LIN {X 0.124,Y -428.626,Z 670.577,A 0.000,B 0.000,C 90.000,E1 103.883} C_DIS
LIN {X -0.109,Y -448.565,Z 670.566,A 0.000,B 0.000,C 90.000,E1 101.827} C_DIS
LIN {X -0.065,Y -469.090,Z 670.555,A 0.000,B 0.000,C 90.000,E1 99.905} C_DIS
LIN {X -0.014,Y -471.282,Z 670.554,A 0.000,B 0.000,C 90.000,E1 99.670} C_DIS
LIN {X -0.163,Y -473.093,Z 670.552,A 0.000,B 0.000,C 90.000,E1 99.434} C_DIS
LIN {X 0.078,Y -474.453,Z 670.551,A 0.000,B 0.000,C 90.000,E1 99.151} C_DIS
LIN {X -0.202,Y -476.161,Z 670.548,A 0.000,B 0.000,C 90.000,E1 98.681} C_DIS
LIN {X -0.076,Y -476.795,Z 670.545,A 0.000,B 0.000,C 90.000,E1 98.163} C_DIS
LIN {X 0.062,Y -476.462,Z 670.542,A 0.000,B 0.000,C 90.000,E1 97.644} C_DIS
LIN {X 0.204,Y -475.113,Z 670.540,A 0.000,B 0.000,C 90.000,E1 97.125} C_DIS
LIN {X 0.067,Y -473.992,Z 670.538,A 0.000,B 0.000,C 90.000,E1 96.891} C_DIS
LIN {X -0.126,Y -472.493,Z 670.537,A 0.000,B 0.000,C 90.000,E1 96.663} C_DIS
LIN {X -0.192,Y -455.641,Z 670.523,A 0.000,B 0.000,C 90.000,E1 94.131} C_DIS
LIN {X 0.189,Y -443.555,Z 670.511,A 0.000,B 0.000,C 90.000,E1 92.007} C_DIS
LIN {X 0.104,Y -433.501,Z 670.501,A 0.000,B 0.000,C 90.000,E1 90.172} C_DIS
LIN {X -0.022,Y -425.963,Z 670.494,A 0.000,B 0.000,C 90.000,E1 88.854} C_DIS
LIN {X -0.041,Y -415.056,Z 670.483,A 0.000,B 0.000,C 90.000,E1 86.963} C_DIS
LIN {X 0.179,Y -404.176,Z 670.472,A 0.000,B 0.000,C 90.000,E1 85.008} C_DIS
LIN {X -0.101,Y -390.407,Z 670.458,A 0.000,B 0.000,C 90.000,E1 82.527} C_DIS
LIN {X 0.116,Y -378.549,Z 670.446,A 0.000,B 0.000,C 90.000,E1 80.208} C_DIS
LIN {X 0.087,Y -365.737,Z 670.431,A 0.000,B 0.000,C 90.000,E1 77.589} C_DIS
LIN {X -0.091,Y -350.683,Z 670.413,A 0.000,B 0.000,C 90.000,E1 74.338} C_DIS
LIN {X -0.019,Y -337.744,Z 670.396,A 0.000,B 0.000,C 90.000,E1 71.275} C_DIS
LIN {X -0.086,Y -323.394,Z 670.375,A 0.000,B 0.000,C 90.000,E1 67.539} C_DIS
LIN {X -0.074,Y -311.579,Z 670.356,A 0.000,B 0.000,C 90.000,E1 64.024} C_DIS
LIN {X -0.193,Y -301.989,Z 670.338,A 0.000,B 0.000,C 90.000,E1 60.795} C_DIS
LIN {X -0.016,Y -293.247,Z 670.319,A 0.000,B 0.000,C 90.000,E1 57.454} C_DIS
LIN {X -0.007,Y -286.662,Z 670.304,A 0.000,B 0.000,C 90.000,E1 54.769} C_DIS
LIN {X -0.067,Y -280.101,Z 670.289,A 0.000,B 0.000,C 90.000,E1 52.065} C_DIS
LIN {X 0.013,Y -274.939,Z 670.278,A 0.000,B 0.000,C 90.000,E1 49.989} C_DIS
LIN {X -0.032,Y -269.443,Z 670.266,A 0.000,B 0.000,C 90.000,E1 47.919} C_DIS
LIN {X 0.004,Y -263.583,Z 670.255,A 0.000,B 0.000,C 90.000,E1 45.810} C_DIS
LIN {X -0.079,Y -257.402,Z 670.243,A 0.000,B 0.000,C 90.000,E1 43.704} C_DIS
LIN {X 0.092,Y -251.028,Z 670.231,A 0.000,B 0.000,C 90.000,E1 41.515} C_DIS
LIN {X 0.007,Y -242.450,Z 670.215,A 0.000,B 0.000,C 90.000,E1 38.624} C_DIS
LIN {X 0.081,Y -232.462,Z 670.194,A 0.000,B 0.000,C 90.000,E1 34.898} C_DIS
LIN {X 0.078,Y -225.134,Z 670.177,A 0.000,B 0.000,C 90.000,E1 31.878} C_DIS
LIN {X 0.042,Y -218.649,Z 670.160,A 0.000,B 0.000,C 90.000,E1 28.821} C_DIS
LIN {X 0.018,Y -212.967,Z 670.143,A 0.000,B 0.000,C 90.000,E1 25.720} C_DIS
LIN {X -0.032,Y -208.075,Z 670.125,A 0.000,B 0.000,C 90.000,E1 22.589} C_DIS
LIN {X 0.022,Y -203.111,Z 670.103,A 0.000,B 0.000,C 90.000,E1 18.598} C_DIS
LIN {X -0.017,Y -199.233,Z 670.081,A 0.000,B 0.000,C 90.000,E1 14.592} C_DIS
LIN {X -0.006,Y -195.919,Z 670.054,A 0.000,B 0.000,C 90.000,E1 9.726} C_DIS
LIN {X 0.082,Y -193.629,Z 670.013,A 0.000,B 0.000,C 90.000,E1 2.350} C_DIS
LIN {X -0.036,Y -195.477,Z 669.961,A 0.000,B 0.000,C 90.000,E1 352.996} C_DIS
LIN {X -0.065,Y -198.507,Z 669.934,A 0.000,B 0.000,C 90.000,E1 348.117} C_DIS
LIN {X 0.026,Y -202.213,Z 669.911,A 0.000,B 0.000,C 90.000,E1 344.047} C_DIS
LIN {X -0.061,Y -206.877,Z 669.889,A 0.000,B 0.000,C 90.000,E1 340.061} C_DIS
LIN {X 0.099,Y -212.320,Z 669.867,A 0.000,B 0.000,C 90.000,E1 336.049} C_DIS
LIN {X 0.007,Y -218.539,Z 669.845,A 0.000,B 0.000,C 90.000,E1 332.153} C_DIS
LIN {X 0.029,Y -225.425,Z 669.824,A 0.000,B 0.000,C 90.000,E1 328.280} C_DIS
LIN {X -0.027,Y -232.928,Z 669.803,A 0.000,B 0.000,C 90.000,E1 324.482} C_DIS
LIN {X 0.003,Y -241.051,Z 669.782,A 0.000,B 0.000,C 90.000,E1 320.723} C_DIS
LIN {X 0.037,Y -250.012,Z 669.761,A 0.000,B 0.000,C 90.000,E1 317.025} C_DIS
LIN {X -0.054,Y -259.057,Z 669.743,A 0.000,B 0.000,C 90.000,E1 313.785} C_DIS
LIN {X 0.029,Y -270.150,Z 669.723,A 0.000,B 0.000,C 90.000,E1 310.216} C_DIS
LIN {X 0.081,Y -281.443,Z 669.706,A 0.000,B 0.000,C 90.000,E1 307.076} C_DIS
LIN {X -0.056,Y -295.332,Z 669.687,A 0.000,B 0.000,C 90.000,E1 303.706} C_DIS
LIN {X 0.006,Y -310.666,Z 669.669,A 0.000,B 0.000,C 90.000,E1 300.384} C_DIS
LIN {X -0.071,Y -327.476,Z 669.651,A 0.000,B 0.000,C 90.000,E1 297.180} C_DIS
LIN {X 0.104,Y -341.711,Z 669.637,A 0.000,B 0.000,C 90.000,E1 294.643} C_DIS
LIN {X 0.144,Y -360.271,Z 669.620,A 0.000,B 0.000,C 90.000,E1 291.589} C_DIS
LIN {X 0.097,Y -372.192,Z 669.610,A 0.000,B 0.000,C 90.000,E1 289.812} C_DIS
LIN {X -0.071,Y -389.779,Z 669.597,A 0.000,B 0.000,C 90.000,E1 287.511} C_DIS
LIN {X -0.123,Y -406.148,Z 669.586,A 0.000,B 0.000,C 90.000,E1 285.536} C_DIS
LIN {X 0.094,Y -417.666,Z 669.578,A 0.000,B 0.000,C 90.000,E1 284.120} C_DIS
LIN {X -0.167,Y -426.483,Z 669.572,A 0.000,B 0.000,C 90.000,E1 283.063} C_DIS
LIN {X -0.137,Y -437.045,Z 669.565,A 0.000,B 0.000,C 90.000,E1 281.715} C_DIS
LIN {X -0.177,Y -445.024,Z 669.559,A 0.000,B 0.000,C 90.000,E1 280.658} C_DIS
LIN {X -0.112,Y -465.214,Z 669.545,A 0.000,B 0.000,C 90.000,E1 278.049} C_DIS
LIN {X -0.217,Y -470.973,Z 669.540,A 0.000,B 0.000,C 90.000,E1 277.296} C_DIS
LIN {X -0.120,Y -474.369,Z 669.538,A 0.000,B 0.000,C 90.000,E1 276.777} C_DIS
LIN {X -0.144,Y -478.628,Z 669.533,A 0.000,B 0.000,C 90.000,E1 276.024} C_DIS
LIN {X -0.047,Y -481.033,Z 669.531,A 0.000,B 0.000,C 90.000,E1 275.511} C_DIS
LIN {X -0.020,Y -483.884,Z 669.526,A 0.000,B 0.000,C 90.000,E1 274.759} C_DIS
LIN {X 0.114,Y -485.270,Z 669.524,A 0.000,B 0.000,C 90.000,E1 274.245} C_DIS
LIN {X -0.187,Y -486.308,Z 669.521,A 0.000,B 0.000,C 90.000,E1 273.784} C_DIS
LIN {X -0.028,Y -486.967,Z 669.518,A 0.000,B 0.000,C 90.000,E1 273.269} C_DIS
LIN {X 0.167,Y -487.304,Z 669.515,A 0.000,B 0.000,C 90.000,E1 272.751} C_DIS
LIN {X -0.146,Y -487.303,Z 669.513,A 0.000,B 0.000,C 90.000,E1 272.293} C_DIS
LIN {X 0.048,Y -487.013,Z 669.510,A 0.000,B 0.000,C 90.000,E1 271.776} C_DIS
LIN {X 0.224,Y -486.400,Z 669.507,A 0.000,B 0.000,C 90.000,E1 271.260} C_DIS
LIN {X -0.086,Y -485.361,Z 669.504,A 0.000,B 0.000,C 90.000,E1 270.802} C_DIS
LIN {X 0.087,Y -483.834,Z 669.502,A 0.000,B 0.000,C 90.000,E1 270.286} C_DIS
LIN {X -0.228,Y -481.687,Z 669.499,A 0.000,B 0.000,C 90.000,E1 269.828} C_DIS
LIN {X -0.070,Y -478.880,Z 669.496,A 0.000,B 0.000,C 90.000,E1 269.312} C_DIS
LIN {X 0.066,Y -475.210,Z 669.493,A 0.000,B 0.000,C 90.000,E1 268.797} C_DIS
LIN {X -0.113,Y -473.058,Z 669.492,A 0.000,B 0.000,C 90.000,E1 268.568} C_DIS
LIN {X 0.039,Y -467.847,Z 669.489,A 0.000,B 0.000,C 90.000,E1 268.051} C_DIS
LIN {X -0.115,Y -464.818,Z 669.488,A 0.000,B 0.000,C 90.000,E1 267.822} C_DIS
LIN {X 0.064,Y -458.384,Z 669.485,A 0.000,B 0.000,C 90.000,E1 267.364} C_DIS
LIN {X -0.102,Y -451.464,Z 669.483,A 0.000,B 0.000,C 90.000,E1 267.020} C_DIS
LIN {X -0.140,Y -444.281,Z 669.482,A 0.000,B 0.000,C 90.000,E1 266.731} C_DIS
LIN {X -0.172,Y -436.408,Z 669.480,A 0.000,B 0.000,C 90.000,E1 266.502} C_DIS
LIN {X -0.153,Y -427.882,Z 669.479,A 0.000,B 0.000,C 90.000,E1 266.331} C_DIS
LIN {X 0.061,Y -420.369,Z 669.479,A 0.000,B 0.000,C 90.000,E1 266.216} C_DIS
LIN {X -0.147,Y -413.980,Z 669.479,A 0.000,B 0.000,C 90.000,E1 266.216} C_DIS
LIN {X -0.086,Y -180.929,Z 669.479,A 0.000,B 0.000,C 90.000,E1 266.216} C_DIS
LIN {X 0.002,Y -180.904,Z 669.474,A 0.000,B 0.000,C 90.000,E1 265.298} C_DIS
LIN {X -0.048,Y -180.244,Z 669.465,A 0.000,B 0.000,C 90.000,E1 263.628} C_DIS
LIN {X -0.029,Y -178.732,Z 669.441,A 0.000,B 0.000,C 90.000,E1 259.398} C_DIS
LIN {X 0.038,Y -175.779,Z 669.413,A 0.000,B 0.000,C 90.000,E1 254.283} C_DIS
LIN {X 0.026,Y -171.963,Z 669.384,A 0.000,B 0.000,C 90.000,E1 249.156} C_DIS
LIN {X 0.063,Y -171.359,Z 669.379,A 0.000,B 0.000,C 90.000,E1 248.284} C_DIS
LIN {X 0.040,Y -167.608,Z 669.355,A 0.000,B 0.000,C 90.000,E1 243.973} C_DIS
LIN {X 0.053,Y -166.255,Z 669.346,A 0.000,B 0.000,C 90.000,E1 242.231} C_DIS
LIN {X 0.040,Y -163.009,Z 669.326,A 0.000,B 0.000,C 90.000,E1 238.742} C_DIS
LIN {X -0.046,Y -160.932,Z 669.312,A 0.000,B 0.000,C 90.000,E1 236.135} C_DIS
LIN {X 0.064,Y -157.692,Z 669.292,A 0.000,B 0.000,C 90.000,E1 232.557} C_DIS
LIN {X 0.001,Y -155.732,Z 669.277,A 0.000,B 0.000,C 90.000,E1 229.908} C_DIS
LIN {X 0.056,Y -151.990,Z 669.252,A 0.000,B 0.000,C 90.000,E1 225.405} C_DIS
LIN {X 0.071,Y -150.234,Z 669.237,A 0.000,B 0.000,C 90.000,E1 222.690} C_DIS
LIN {X -0.006,Y -146.995,Z 669.212,A 0.000,B 0.000,C 90.000,E1 218.177} C_DIS
LIN {X -0.016,Y -145.580,Z 669.197,A 0.000,B 0.000,C 90.000,E1 215.438} C_DIS
LIN {X -0.022,Y -142.969,Z 669.171,A 0.000,B 0.000,C 90.000,E1 210.846} C_DIS
LIN {X 0.032,Y -141.596,Z 669.151,A 0.000,B 0.000,C 90.000,E1 207.129} C_DIS
LIN {X -0.052,Y -139.422,Z 669.115,A 0.000,B 0.000,C 90.000,E1 200.663} C_DIS
LIN {X -0.001,Y -139.149,Z 669.104,A 0.000,B 0.000,C 90.000,E1 198.779} C_DIS
LIN {X 0.021,Y -138.346,Z 669.058,A 0.000,B 0.000,C 90.000,E1 190.366} C_DIS
LIN {X 0.006,Y -139.487,Z 669.006,A 0.000,B 0.000,C 90.000,E1 181.031} C_DIS
LIN {X -0.054,Y -141.088,Z 668.975,A 0.000,B 0.000,C 90.000,E1 175.469} C_DIS
LIN {X 0.041,Y -142.466,Z 668.959,A 0.000,B 0.000,C 90.000,E1 172.648} C_DIS
LIN {X -0.011,Y -144.711,Z 668.934,A 0.000,B 0.000,C 90.000,E1 168.049} C_DIS
LIN {X -0.060,Y -147.309,Z 668.913,A 0.000,B 0.000,C 90.000,E1 164.393} C_DIS
LIN {X -0.045,Y -150.631,Z 668.888,A 0.000,B 0.000,C 90.000,E1 159.826} C_DIS
LIN {X 0.031,Y -154.107,Z 668.868,A 0.000,B 0.000,C 90.000,E1 156.177} C_DIS
LIN {X -0.045,Y -157.530,Z 668.848,A 0.000,B 0.000,C 90.000,E1 152.615} C_DIS
LIN {X -0.100,Y -161.766,Z 668.828,A 0.000,B 0.000,C 90.000,E1 149.076} C_DIS
LIN {X 0.005,Y -165.958,Z 668.808,A 0.000,B 0.000,C 90.000,E1 145.515} C_DIS
LIN {X 0.001,Y -170.952,Z 668.789,A 0.000,B 0.000,C 90.000,E1 142.029} C_DIS
LIN {X 0.053,Y -175.820,Z 668.770,A 0.000,B 0.000,C 90.000,E1 138.566} C_DIS
LIN {X 0.048,Y -181.427,Z 668.751,A 0.000,B 0.000,C 90.000,E1 135.162} C_DIS
LIN {X -0.078,Y -186.932,Z 668.732,A 0.000,B 0.000,C 90.000,E1 131.838} C_DIS
LIN {X 0.094,Y -191.070,Z 668.720,A 0.000,B 0.000,C 90.000,E1 129.564} C_DIS
LIN {X 0.096,Y -288.280,Z 668.720,A 0.000,B 0.000,C 90.000,E1 129.564} C_DIS
LIN {X -0.042,Y -290.385,Z 668.720,A 0.000,B 0.000,C 90.000,E1 129.564} C_DIS
LIN {X -0.007,Y -295.282,Z 668.718,A 0.000,B 0.000,C 90.000,E1 129.322} C_DIS
LIN {X -0.071,Y -298.456,Z 668.717,A 0.000,B 0.000,C 90.000,E1 129.036} C_DIS
LIN {X 0.096,Y -302.112,Z 668.714,A 0.000,B 0.000,C 90.000,E1 128.463} C_DIS
LIN {X -0.144,Y -303.684,Z 668.712,A 0.000,B 0.000,C 90.000,E1 128.177} C_DIS
LIN {X 0.042,Y -304.919,Z 668.710,A 0.000,B 0.000,C 90.000,E1 127.810} C_DIS
LIN {X -0.050,Y -316.534,Z 668.688,A 0.000,B 0.000,C 90.000,E1 123.913} C_DIS
LIN {X 0.130,Y -326.607,Z 668.672,A 0.000,B 0.000,C 90.000,E1 121.003} C_DIS
LIN {X -0.186,Y -338.014,Z 668.657,A 0.000,B 0.000,C 90.000,E1 118.231} C_DIS
LIN {X 0.109,Y -350.850,Z 668.641,A 0.000,B 0.000,C 90.000,E1 115.412} C_DIS
LIN {X -0.052,Y -363.556,Z 668.628,A 0.000,B 0.000,C 90.000,E1 113.025} C_DIS
LIN {X -0.049,Y -377.574,Z 668.615,A 0.000,B 0.000,C 90.000,E1 110.663} C_DIS
LIN {X -0.100,Y -393.007,Z 668.602,A 0.000,B 0.000,C 90.000,E1 108.362} C_DIS
LIN {X 0.119,Y -409.967,Z 668.589,A 0.000,B 0.000,C 90.000,E1 106.079} C_DIS
LIN {X 0.141,Y -428.577,Z 668.577,A 0.000,B 0.000,C 90.000,E1 103.883} C_DIS
LIN {X -0.093,Y -448.516,Z 668.566,A 0.000,B 0.000,C 90.000,E1 101.827} C_DIS
LIN {X -0.051,Y -469.041,Z 668.555,A 0.000,B 0.000,C 90.000,E1 99.905} C_DIS
LIN {X -0.001,Y -471.263,Z 668.554,A 0.000,B 0.000,C 90.000,E1 99.670} C_DIS
LIN {X -0.137,Y -473.086,Z 668.552,A 0.000,B 0.000,C 90.000,E1 99.434} C_DIS
LIN {X 0.118,Y -474.458,Z 668.551,A 0.000,B 0.000,C 90.000,E1 99.151} C_DIS
LIN {X -0.162,Y -476.198,Z 668.548,A 0.000,B 0.000,C 90.000,E1 98.681} C_DIS
LIN {X -0.036,Y -476.858,Z 668.545,A 0.000,B 0.000,C 90.000,E1 98.163} C_DIS
LIN {X 0.102,Y -476.549,Z 668.543,A 0.000,B 0.000,C 90.000,E1 97.644} C_DIS
LIN {X -0.227,Y -475.228,Z 668.540,A 0.000,B 0.000,C 90.000,E1 97.182} C_DIS
LIN {X 0.108,Y -474.123,Z 668.538,A 0.000,B 0.000,C 90.000,E1 96.891} C_DIS
LIN {X -0.084,Y -472.648,Z 668.537,A 0.000,B 0.000,C 90.000,E1 96.663} C_DIS
LIN {X -0.148,Y -455.789,Z 668.523,A 0.000,B 0.000,C 90.000,E1 94.131} C_DIS
LIN {X 0.038,Y -445.138,Z 668.513,A 0.000,B 0.000,C 90.000,E1 92.293} C_DIS
LIN {X 0.150,Y -433.624,Z 668.501,A 0.000,B 0.000,C 90.000,E1 90.172} C_DIS
LIN {X 0.025,Y -426.101,Z 668.494,A 0.000,B 0.000,C 90.000,E1 88.854} C_DIS
LIN {X 0.128,Y -413.658,Z 668.482,A 0.000,B 0.000,C 90.000,E1 86.674} C_DIS
LIN {X -0.119,Y -402.761,Z 668.471,A 0.000,B 0.000,C 90.000,E1 84.780} C_DIS
LIN {X -0.042,Y -389.067,Z 668.457,A 0.000,B 0.000,C 90.000,E1 82.243} C_DIS
LIN {X 0.131,Y -377.270,Z 668.444,A 0.000,B 0.000,C 90.000,E1 79.926} C_DIS
LIN {X 0.145,Y -365.905,Z 668.431,A 0.000,B 0.000,C 90.000,E1 77.589} C_DIS
LIN {X 0.004,Y -349.580,Z 668.411,A 0.000,B 0.000,C 90.000,E1 74.031} C_DIS
LIN {X -0.073,Y -335.511,Z 668.393,A 0.000,B 0.000,C 90.000,E1 70.678} C_DIS
LIN {X -0.105,Y -321.395,Z 668.372,A 0.000,B 0.000,C 90.000,E1 66.922} C_DIS
LIN {X -0.023,Y -309.848,Z 668.352,A 0.000,B 0.000,C 90.000,E1 63.384} C_DIS
LIN {X -0.051,Y -300.429,Z 668.334,A 0.000,B 0.000,C 90.000,E1 60.127} C_DIS
LIN {X 0.073,Y -291.830,Z 668.316,A 0.000,B 0.000,C 90.000,E1 56.786} C_DIS
LIN {X -0.029,Y -285.272,Z 668.301,A 0.000,B 0.000,C 90.000,E1 54.116} C_DIS
LIN {X 0.029,Y -280.380,Z 668.289,A 0.000,B 0.000,C 90.000,E1 52.065} C_DIS
LIN {X 0.113,Y -275.230,Z 668.278,A 0.000,B 0.000,C 90.000,E1 49.989} C_DIS
LIN {X 0.073,Y -269.749,Z 668.266,A 0.000,B 0.000,C 90.000,E1 47.919} C_DIS
LIN {X 0.112,Y -263.900,Z 668.255,A 0.000,B 0.000,C 90.000,E1 45.810} C_DIS
LIN {X 0.033,Y -257.707,Z 668.243,A 0.000,B 0.000,C 90.000,E1 43.704} C_DIS
LIN {X 0.039,Y -251.286,Z 668.231,A 0.000,B 0.000,C 90.000,E1 41.553} C_DIS
LIN {X -0.066,Y -242.697,Z 668.215,A 0.000,B 0.000,C 90.000,E1 38.669} C_DIS
LIN {X 0.070,Y -234.636,Z 668.198,A 0.000,B 0.000,C 90.000,E1 35.678} C_DIS
LIN {X 0.058,Y -227.139,Z 668.182,A 0.000,B 0.000,C 90.000,E1 32.673} C_DIS
LIN {X 0.067,Y -220.415,Z 668.165,A 0.000,B 0.000,C 90.000,E1 29.617} C_DIS
LIN {X -0.004,Y -214.533,Z 668.147,A 0.000,B 0.000,C 90.000,E1 26.539} C_DIS
LIN {X 0.064,Y -209.445,Z 668.130,A 0.000,B 0.000,C 90.000,E1 23.387} C_DIS
LIN {X -0.041,Y -205.146,Z 668.112,A 0.000,B 0.000,C 90.000,E1 20.248} C_DIS
LIN {X -0.084,Y -200.824,Z 668.090,A 0.000,B 0.000,C 90.000,E1 16.260} C_DIS
LIN {X 0.079,Y -197.041,Z 668.063,A 0.000,B 0.000,C 90.000,E1 11.366} C_DIS
LIN {X 0.021,Y -194.359,Z 668.032,A 0.000,B 0.000,C 90.000,E1 5.682} C_DIS
LIN {X -0.032,Y -195.570,Z 667.961,A 0.000,B 0.000,C 90.000,E1 352.996} C_DIS
LIN {X -0.057,Y -198.573,Z 667.934,A 0.000,B 0.000,C 90.000,E1 348.117} C_DIS
LIN {X 0.035,Y -202.276,Z 667.911,A 0.000,B 0.000,C 90.000,E1 344.047} C_DIS
LIN {X -0.049,Y -206.944,Z 667.889,A 0.000,B 0.000,C 90.000,E1 340.061} C_DIS
LIN {X -0.081,Y -212.381,Z 667.867,A 0.000,B 0.000,C 90.000,E1 336.102} C_DIS
LIN {X 0.024,Y -218.597,Z 667.845,A 0.000,B 0.000,C 90.000,E1 332.153} C_DIS
LIN {X 0.048,Y -225.472,Z 667.824,A 0.000,B 0.000,C 90.000,E1 328.280} C_DIS
LIN {X -0.006,Y -232.961,Z 667.803,A 0.000,B 0.000,C 90.000,E1 324.482} C_DIS
LIN {X 0.027,Y -241.067,Z 667.782,A 0.000,B 0.000,C 90.000,E1 320.723} C_DIS
LIN {X -0.121,Y -250.016,Z 667.761,A 0.000,B 0.000,C 90.000,E1 317.067} C_DIS
LIN {X -0.029,Y -259.023,Z 667.743,A 0.000,B 0.000,C 90.000,E1 313.785} C_DIS
LIN {X -0.120,Y -270.113,Z 667.724,A 0.000,B 0.000,C 90.000,E1 310.253} C_DIS
LIN {X 0.107,Y -281.406,Z 667.706,A 0.000,B 0.000,C 90.000,E1 307.076} C_DIS
LIN {X -0.031,Y -295.266,Z 667.687,A 0.000,B 0.000,C 90.000,E1 303.706} C_DIS
LIN {X 0.031,Y -310.630,Z 667.669,A 0.000,B 0.000,C 90.000,E1 300.384} C_DIS
LIN {X -0.046,Y -327.436,Z 667.651,A 0.000,B 0.000,C 90.000,E1 297.180} C_DIS
LIN {X 0.129,Y -341.626,Z 667.637,A 0.000,B 0.000,C 90.000,E1 294.643} C_DIS
LIN {X 0.167,Y -360.172,Z 667.620,A 0.000,B 0.000,C 90.000,E1 291.589} C_DIS
LIN {X 0.118,Y -372.082,Z 667.610,A 0.000,B 0.000,C 90.000,E1 289.812} C_DIS
LIN {X -0.185,Y -387.358,Z 667.599,A 0.000,B 0.000,C 90.000,E1 287.819} C_DIS
LIN {X -0.106,Y -406.022,Z 667.586,A 0.000,B 0.000,C 90.000,E1 285.536} C_DIS
LIN {X 0.110,Y -417.537,Z 667.579,A 0.000,B 0.000,C 90.000,E1 284.120} C_DIS
LIN {X -0.152,Y -426.371,Z 667.572,A 0.000,B 0.000,C 90.000,E1 283.063} C_DIS
LIN {X -0.123,Y -436.911,Z 667.565,A 0.000,B 0.000,C 90.000,E1 281.715} C_DIS
LIN {X -0.164,Y -444.894,Z 667.559,A 0.000,B 0.000,C 90.000,E1 280.658} C_DIS
LIN {X -0.136,Y -460.983,Z 667.547,A 0.000,B 0.000,C 90.000,E1 278.568} C_DIS
LIN {X 0.185,Y -467.176,Z 667.543,A 0.000,B 0.000,C 90.000,E1 277.757} C_DIS
LIN {X 0.104,Y -472.664,Z 667.539,A 0.000,B 0.000,C 90.000,E1 277.004} C_DIS
LIN {X 0.211,Y -475.802,Z 667.536,A 0.000,B 0.000,C 90.000,E1 276.486} C_DIS
LIN {X 0.147,Y -479.798,Z 667.532,A 0.000,B 0.000,C 90.000,E1 275.739} C_DIS
LIN {X -0.179,Y -482.029,Z 667.529,A 0.000,B 0.000,C 90.000,E1 275.277} C_DIS
LIN {X -0.013,Y -483.827,Z 667.526,A 0.000,B 0.000,C 90.000,E1 274.759} C_DIS
LIN {X 0.122,Y -485.229,Z 667.524,A 0.000,B 0.000,C 90.000,E1 274.245} C_DIS
LIN {X -0.180,Y -486.256,Z 667.521,A 0.000,B 0.000,C 90.000,E1 273.784} C_DIS
LIN {X -0.020,Y -486.938,Z 667.518,A 0.000,B 0.000,C 90.000,E1 273.269} C_DIS
LIN {X 0.174,Y -487.249,Z 667.515,A 0.000,B 0.000,C 90.000,E1 272.751} C_DIS
LIN {X -0.139,Y -487.282,Z 667.513,A 0.000,B 0.000,C 90.000,E1 272.293} C_DIS
LIN {X 0.054,Y -486.979,Z 667.510,A 0.000,B 0.000,C 90.000,E1 271.776} C_DIS
LIN {X 0.230,Y -486.357,Z 667.507,A 0.000,B 0.000,C 90.000,E1 271.260} C_DIS
LIN {X -0.080,Y -485.336,Z 667.504,A 0.000,B 0.000,C 90.000,E1 270.802} C_DIS
LIN {X 0.093,Y -483.816,Z 667.502,A 0.000,B 0.000,C 90.000,E1 270.286} C_DIS
LIN {X -0.223,Y -481.716,Z 667.499,A 0.000,B 0.000,C 90.000,E1 269.828} C_DIS
LIN {X -0.065,Y -478.903,Z 667.496,A 0.000,B 0.000,C 90.000,E1 269.312} C_DIS
LIN {X -0.235,Y -477.219,Z 667.495,A 0.000,B 0.000,C 90.000,E1 269.083} C_DIS
LIN {X -0.108,Y -473.115,Z 667.492,A 0.000,B 0.000,C 90.000,E1 268.568} C_DIS
LIN {X 0.052,Y -467.906,Z 667.489,A 0.000,B 0.000,C 90.000,E1 268.051} C_DIS
LIN {X -0.095,Y -464.881,Z 667.488,A 0.000,B 0.000,C 90.000,E1 267.822} C_DIS
LIN {X 0.089,Y -458.526,Z 667.485,A 0.000,B 0.000,C 90.000,E1 267.364} C_DIS
LIN {X -0.103,Y -451.603,Z 667.483,A 0.000,B 0.000,C 90.000,E1 267.020} C_DIS
LIN {X -0.170,Y -444.240,Z 667.482,A 0.000,B 0.000,C 90.000,E1 266.731} C_DIS
LIN {X -0.183,Y -440.751,Z 667.481,A 0.000,B 0.000,C 90.000,E1 266.617} C_DIS
LIN {X 0.048,Y -432.707,Z 667.480,A 0.000,B 0.000,C 90.000,E1 266.388} C_DIS
LIN {X -0.148,Y -423.635,Z 667.479,A 0.000,B 0.000,C 90.000,E1 266.274} C_DIS
LIN {X -0.155,Y -414.628,Z 667.479,A 0.000,B 0.000,C 90.000,E1 266.216} C_DIS
LIN {X -0.090,Y -180.929,Z 667.479,A 0.000,B 0.000,C 90.000,E1 266.216} C_DIS
LIN {X -0.008,Y -180.903,Z 667.474,A 0.000,B 0.000,C 90.000,E1 265.298} C_DIS
LIN {X -0.058,Y -180.243,Z 667.464,A 0.000,B 0.000,C 90.000,E1 263.628} C_DIS
LIN {X -0.039,Y -178.729,Z 667.441,A 0.000,B 0.000,C 90.000,E1 259.398} C_DIS
LIN {X 0.029,Y -175.778,Z 667.413,A 0.000,B 0.000,C 90.000,E1 254.283} C_DIS
LIN {X 0.016,Y -171.961,Z 667.384,A 0.000,B 0.000,C 90.000,E1 249.156} C_DIS
LIN {X 0.053,Y -171.356,Z 667.379,A 0.000,B 0.000,C 90.000,E1 248.284} C_DIS
LIN {X 0.031,Y -167.606,Z 667.355,A 0.000,B 0.000,C 90.000,E1 243.973} C_DIS
LIN {X 0.044,Y -166.252,Z 667.346,A 0.000,B 0.000,C 90.000,E1 242.231} C_DIS
LIN {X 0.032,Y -163.006,Z 667.326,A 0.000,B 0.000,C 90.000,E1 238.742} C_DIS
LIN {X 0.078,Y -160.929,Z 667.312,A 0.000,B 0.000,C 90.000,E1 236.087} C_DIS
LIN {X 0.055,Y -157.690,Z 667.292,A 0.000,B 0.000,C 90.000,E1 232.557} C_DIS
LIN {X -0.007,Y -155.729,Z 667.277,A 0.000,B 0.000,C 90.000,E1 229.908} C_DIS
LIN {X 0.047,Y -151.988,Z 667.252,A 0.000,B 0.000,C 90.000,E1 225.405} C_DIS
LIN {X 0.063,Y -150.232,Z 667.237,A 0.000,B 0.000,C 90.000,E1 222.690} C_DIS
LIN {X -0.015,Y -146.993,Z 667.212,A 0.000,B 0.000,C 90.000,E1 218.177} C_DIS
LIN {X -0.024,Y -145.578,Z 667.197,A 0.000,B 0.000,C 90.000,E1 215.438} C_DIS
LIN {X -0.030,Y -142.967,Z 667.171,A 0.000,B 0.000,C 90.000,E1 210.846} C_DIS
LIN {X 0.023,Y -141.594,Z 667.151,A 0.000,B 0.000,C 90.000,E1 207.129} C_DIS
LIN {X 0.069,Y -139.420,Z 667.115,A 0.000,B 0.000,C 90.000,E1 200.610} C_DIS
LIN {X -0.010,Y -139.148,Z 667.104,A 0.000,B 0.000,C 90.000,E1 198.779} C_DIS
LIN {X 0.012,Y -138.345,Z 667.058,A 0.000,B 0.000,C 90.000,E1 190.366} C_DIS
LIN {X -0.002,Y -139.488,Z 667.006,A 0.000,B 0.000,C 90.000,E1 181.031} C_DIS
LIN {X -0.061,Y -141.090,Z 666.975,A 0.000,B 0.000,C 90.000,E1 175.469} C_DIS
LIN {X 0.033,Y -142.467,Z 666.959,A 0.000,B 0.000,C 90.000,E1 172.648} C_DIS
LIN {X -0.020,Y -144.713,Z 666.934,A 0.000,B 0.000,C 90.000,E1 168.049} C_DIS
LIN {X -0.068,Y -147.312,Z 666.913,A 0.000,B 0.000,C 90.000,E1 164.393} C_DIS
LIN {X -0.053,Y -150.633,Z 666.888,A 0.000,B 0.000,C 90.000,E1 159.826} C_DIS
LIN {X 0.022,Y -154.109,Z 666.868,A 0.000,B 0.000,C 90.000,E1 156.177} C_DIS
LIN {X -0.054,Y -157.534,Z 666.848,A 0.000,B 0.000,C 90.000,E1 152.615} C_DIS
LIN {X -0.028,Y -161.770,Z 666.828,A 0.000,B 0.000,C 90.000,E1 149.046} C_DIS
LIN {X -0.004,Y -165.963,Z 666.808,A 0.000,B 0.000,C 90.000,E1 145.515} C_DIS
LIN {X -0.008,Y -170.956,Z 666.789,A 0.000,B 0.000,C 90.000,E1 142.029} C_DIS
LIN {X 0.044,Y -175.825,Z 666.770,A 0.000,B 0.000,C 90.000,E1 138.566} C_DIS
LIN {X 0.038,Y -181.432,Z 666.751,A 0.000,B 0.000,C 90.000,E1 135.162} C_DIS
LIN {X -0.087,Y -186.937,Z 666.732,A 0.000,B 0.000,C 90.000,E1 131.838} C_DIS
LIN {X 0.083,Y -191.075,Z 666.720,A 0.000,B 0.000,C 90.000,E1 129.564} C_DIS
LIN {X 0.082,Y -288.955,Z 666.720,A 0.000,B 0.000,C 90.000,E1 129.564} C_DIS
LIN {X -0.056,Y -290.538,Z 666.720,A 0.000,B 0.000,C 90.000,E1 129.564} C_DIS
LIN {X -0.023,Y -295.318,Z 666.718,A 0.000,B 0.000,C 90.000,E1 129.322} C_DIS
LIN {X 0.109,Y -298.532,Z 666.717,A 0.000,B 0.000,C 90.000,E1 128.991} C_DIS
LIN {X 0.018,Y -302.175,Z 666.714,A 0.000,B 0.000,C 90.000,E1 128.463} C_DIS
LIN {X -0.034,Y -303.727,Z 666.712,A 0.000,B 0.000,C 90.000,E1 128.141} C_DIS
LIN {X -0.036,Y -304.948,Z 666.710,A 0.000,B 0.000,C 90.000,E1 127.810} C_DIS
LIN {X -0.130,Y -316.559,Z 666.688,A 0.000,B 0.000,C 90.000,E1 123.913} C_DIS
LIN {X 0.049,Y -326.640,Z 666.672,A 0.000,B 0.000,C 90.000,E1 121.003} C_DIS
LIN {X 0.028,Y -338.053,Z 666.657,A 0.000,B 0.000,C 90.000,E1 118.180} C_DIS
LIN {X 0.024,Y -350.896,Z 666.641,A 0.000,B 0.000,C 90.000,E1 115.412} C_DIS
LIN {X -0.139,Y -363.609,Z 666.628,A 0.000,B 0.000,C 90.000,E1 113.025} C_DIS
LIN {X -0.138,Y -377.635,Z 666.615,A 0.000,B 0.000,C 90.000,E1 110.663} C_DIS
LIN {X -0.191,Y -393.076,Z 666.602,A 0.000,B 0.000,C 90.000,E1 108.362} C_DIS
LIN {X 0.026,Y -410.045,Z 666.589,A 0.000,B 0.000,C 90.000,E1 106.079} C_DIS
LIN {X 0.045,Y -428.665,Z 666.577,A 0.000,B 0.000,C 90.000,E1 103.883} C_DIS
LIN {X -0.187,Y -448.608,Z 666.566,A 0.000,B 0.000,C 90.000,E1 101.827} C_DIS
LIN {X -0.142,Y -469.136,Z 666.555,A 0.000,B 0.000,C 90.000,E1 99.905} C_DIS
LIN {X -0.091,Y -471.351,Z 666.554,A 0.000,B 0.000,C 90.000,E1 99.670} C_DIS
LIN {X 0.236,Y -473.173,Z 666.552,A 0.000,B 0.000,C 90.000,E1 99.378} C_DIS
LIN {X 0.020,Y -474.542,Z 666.551,A 0.000,B 0.000,C 90.000,E1 99.151} C_DIS
LIN {X 0.212,Y -476.277,Z 666.548,A 0.000,B 0.000,C 90.000,E1 98.624} C_DIS
LIN {X -0.133,Y -476.934,Z 666.545,A 0.000,B 0.000,C 90.000,E1 98.163} C_DIS
LIN {X 0.005,Y -476.621,Z 666.542,A 0.000,B 0.000,C 90.000,E1 97.644} C_DIS
LIN {X 0.149,Y -475.296,Z 666.540,A 0.000,B 0.000,C 90.000,E1 97.125} C_DIS
LIN {X 0.013,Y -474.189,Z 666.538,A 0.000,B 0.000,C 90.000,E1 96.891} C_DIS
LIN {X -0.179,Y -472.707,Z 666.537,A 0.000,B 0.000,C 90.000,E1 96.663} C_DIS
LIN {X -0.239,Y -455.834,Z 666.523,A 0.000,B 0.000,C 90.000,E1 94.131} C_DIS
LIN {X -0.049,Y -445.176,Z 666.513,A 0.000,B 0.000,C 90.000,E1 92.293} C_DIS
LIN {X -0.093,Y -435.108,Z 666.503,A 0.000,B 0.000,C 90.000,E1 90.458} C_DIS
LIN {X -0.196,Y -427.678,Z 666.495,A 0.000,B 0.000,C 90.000,E1 89.141} C_DIS
LIN {X -0.169,Y -416.798,Z 666.485,A 0.000,B 0.000,C 90.000,E1 87.249} C_DIS
LIN {X -0.007,Y -407.480,Z 666.475,A 0.000,B 0.000,C 90.000,E1 85.584} C_DIS
LIN {X 0.144,Y -393.642,Z 666.462,A 0.000,B 0.000,C 90.000,E1 83.053} C_DIS
LIN {X 0.079,Y -380.258,Z 666.447,A 0.000,B 0.000,C 90.000,E1 80.500} C_DIS
LIN {X 0.093,Y -367.391,Z 666.433,A 0.000,B 0.000,C 90.000,E1 77.881} C_DIS
LIN {X -0.062,Y -353.623,Z 666.416,A 0.000,B 0.000,C 90.000,E1 74.936} C_DIS
LIN {X 0.079,Y -343.186,Z 666.403,A 0.000,B 0.000,C 90.000,E1 72.489} C_DIS
LIN {X 0.131,Y -330.795,Z 666.386,A 0.000,B 0.000,C 90.000,E1 69.390} C_DIS
LIN {X 0.112,Y -318.276,Z 666.366,A 0.000,B 0.000,C 90.000,E1 65.921} C_DIS
LIN {X -0.146,Y -306.174,Z 666.345,A 0.000,B 0.000,C 90.000,E1 62.103} C_DIS
LIN {X 0.009,Y -297.099,Z 666.327,A 0.000,B 0.000,C 90.000,E1 58.791} C_DIS
LIN {X -0.060,Y -288.742,Z 666.308,A 0.000,B 0.000,C 90.000,E1 55.468} C_DIS
LIN {X -0.065,Y -282.220,Z 666.293,A 0.000,B 0.000,C 90.000,E1 52.763} C_DIS
LIN {X -0.114,Y -277.216,Z 666.282,A 0.000,B 0.000,C 90.000,E1 50.723} C_DIS
LIN {X 0.092,Y -271.861,Z 666.270,A 0.000,B 0.000,C 90.000,E1 48.609} C_DIS
LIN {X -0.011,Y -266.113,Z 666.259,A 0.000,B 0.000,C 90.000,E1 46.539} C_DIS
LIN {X -0.046,Y -260.029,Z 666.247,A 0.000,B 0.000,C 90.000,E1 44.433} C_DIS
LIN {X -0.011,Y -253.648,Z 666.235,A 0.000,B 0.000,C 90.000,E1 42.285} C_DIS
LIN {X 0.107,Y -247.163,Z 666.223,A 0.000,B 0.000,C 90.000,E1 40.092} C_DIS
LIN {X 0.115,Y -238.763,Z 666.207,A 0.000,B 0.000,C 90.000,E1 37.156} C_DIS
LIN {X 0.015,Y -230.983,Z 666.190,A 0.000,B 0.000,C 90.000,E1 34.199} C_DIS
LIN {X -0.027,Y -223.852,Z 666.173,A 0.000,B 0.000,C 90.000,E1 31.180} C_DIS
LIN {X -0.015,Y -217.538,Z 666.156,A 0.000,B 0.000,C 90.000,E1 28.103} C_DIS
LIN {X 0.034,Y -212.061,Z 666.139,A 0.000,B 0.000,C 90.000,E1 24.975} C_DIS
LIN {X -0.036,Y -207.362,Z 666.121,A 0.000,B 0.000,C 90.000,E1 21.844} C_DIS
LIN {X -0.074,Y -202.596,Z 666.099,A 0.000,B 0.000,C 90.000,E1 17.873} C_DIS
LIN {X 0.010,Y -198.909,Z 666.077,A 0.000,B 0.000,C 90.000,E1 13.828} C_DIS
LIN {X -0.027,Y -195.750,Z 666.050,A 0.000,B 0.000,C 90.000,E1 8.973} C_DIS
LIN {X -0.035,Y -193.789,Z 665.997,A 0.000,B 0.000,C 90.000,E1 359.542} C_DIS
LIN {X -0.048,Y -196.027,Z 665.956,A 0.000,B 0.000,C 90.000,E1 352.186} C_DIS
LIN {X -0.019,Y -199.320,Z 665.929,A 0.000,B 0.000,C 90.000,E1 347.297} C_DIS
LIN {X -0.046,Y -203.192,Z 665.907,A 0.000,B 0.000,C 90.000,E1 343.268} C_DIS
LIN {X -0.033,Y -208.033,Z 665.885,A 0.000,B 0.000,C 90.000,E1 339.263} C_DIS
LIN {X 0.055,Y -213.626,Z 665.863,A 0.000,B 0.000,C 90.000,E1 335.281} C_DIS
LIN {X 0.005,Y -219.977,Z 665.841,A 0.000,B 0.000,C 90.000,E1 331.385} C_DIS
LIN {X -0.012,Y -226.982,Z 665.820,A 0.000,B 0.000,C 90.000,E1 327.533} C_DIS
LIN {X 0.114,Y -234.569,Z 665.799,A 0.000,B 0.000,C 90.000,E1 323.703} C_DIS
LIN {X 0.010,Y -242.810,Z 665.778,A 0.000,B 0.000,C 90.000,E1 319.989} C_DIS
LIN {X 0.081,Y -251.936,Z 665.757,A 0.000,B 0.000,C 90.000,E1 316.296} C_DIS
LIN {X 0.094,Y -262.186,Z 665.737,A 0.000,B 0.000,C 90.000,E1 312.690} C_DIS
LIN {X -0.150,Y -272.473,Z 665.720,A 0.000,B 0.000,C 90.000,E1 309.564} C_DIS
LIN {X -0.077,Y -285.357,Z 665.700,A 0.000,B 0.000,C 90.000,E1 306.091} C_DIS
LIN {X -0.014,Y -298.151,Z 665.684,A 0.000,B 0.000,C 90.000,E1 303.038} C_DIS
LIN {X -0.009,Y -313.824,Z 665.665,A 0.000,B 0.000,C 90.000,E1 299.745} C_DIS
LIN {X -0.075,Y -329.133,Z 665.649,A 0.000,B 0.000,C 90.000,E1 296.873} C_DIS
LIN {X 0.152,Y -341.516,Z 665.637,A 0.000,B 0.000,C 90.000,E1 294.643} C_DIS
LIN {X 0.142,Y -358.161,Z 665.622,A 0.000,B 0.000,C 90.000,E1 291.897} C_DIS
LIN {X 0.056,Y -369.871,Z 665.612,A 0.000,B 0.000,C 90.000,E1 290.120} C_DIS
LIN {X 0.186,Y -384.978,Z 665.600,A 0.000,B 0.000,C 90.000,E1 288.055} C_DIS
LIN {X 0.110,Y -403.548,Z 665.588,A 0.000,B 0.000,C 90.000,E1 285.788} C_DIS
LIN {X 0.010,Y -415.141,Z 665.580,A 0.000,B 0.000,C 90.000,E1 284.411} C_DIS
LIN {X 0.127,Y -424.082,Z 665.574,A 0.000,B 0.000,C 90.000,E1 283.300} C_DIS
LIN {X 0.124,Y -434.733,Z 665.566,A 0.000,B 0.000,C 90.000,E1 281.951} C_DIS
LIN {X 0.064,Y -442.844,Z 665.561,A 0.000,B 0.000,C 90.000,E1 280.894} C_DIS
LIN {X 0.055,Y -458.820,Z 665.549,A 0.000,B 0.000,C 90.000,E1 278.803} C_DIS
LIN {X 0.193,Y -467.127,Z 665.543,A 0.000,B 0.000,C 90.000,E1 277.757} C_DIS
LIN {X -0.199,Y -470.910,Z 665.540,A 0.000,B 0.000,C 90.000,E1 277.296} C_DIS
LIN {X -0.103,Y -474.279,Z 665.538,A 0.000,B 0.000,C 90.000,E1 276.777} C_DIS
LIN {X -0.128,Y -478.499,Z 665.533,A 0.000,B 0.000,C 90.000,E1 276.024} C_DIS
LIN {X -0.171,Y -481.960,Z 665.529,A 0.000,B 0.000,C 90.000,E1 275.277} C_DIS
LIN {X -0.006,Y -483.802,Z 665.526,A 0.000,B 0.000,C 90.000,E1 274.759} C_DIS
LIN {X 0.128,Y -485.200,Z 665.524,A 0.000,B 0.000,C 90.000,E1 274.245} C_DIS
LIN {X -0.173,Y -486.235,Z 665.521,A 0.000,B 0.000,C 90.000,E1 273.784} C_DIS
LIN {X -0.014,Y -486.865,Z 665.518,A 0.000,B 0.000,C 90.000,E1 273.269} C_DIS
LIN {X 0.180,Y -487.204,Z 665.515,A 0.000,B 0.000,C 90.000,E1 272.751} C_DIS
LIN {X -0.134,Y -487.252,Z 665.513,A 0.000,B 0.000,C 90.000,E1 272.293} C_DIS
LIN {X 0.060,Y -486.952,Z 665.510,A 0.000,B 0.000,C 90.000,E1 271.776} C_DIS
LIN {X 0.235,Y -486.329,Z 665.507,A 0.000,B 0.000,C 90.000,E1 271.260} C_DIS
LIN {X -0.075,Y -485.286,Z 665.504,A 0.000,B 0.000,C 90.000,E1 270.802} C_DIS
LIN {X 0.098,Y -483.745,Z 665.502,A 0.000,B 0.000,C 90.000,E1 270.286} C_DIS
LIN {X -0.218,Y -481.719,Z 665.499,A 0.000,B 0.000,C 90.000,E1 269.828} C_DIS
LIN {X -0.061,Y -478.891,Z 665.496,A 0.000,B 0.000,C 90.000,E1 269.312} C_DIS
LIN {X -0.230,Y -477.255,Z 665.495,A 0.000,B 0.000,C 90.000,E1 269.083} C_DIS
LIN {X -0.103,Y -473.139,Z 665.492,A 0.000,B 0.000,C 90.000,E1 268.568} C_DIS
LIN {X 0.052,Y -467.949,Z 665.489,A 0.000,B 0.000,C 90.000,E1 268.051} C_DIS
LIN {X -0.008,Y -461.940,Z 665.487,A 0.000,B 0.000,C 90.000,E1 267.593} C_DIS
LIN {X 0.081,Y -458.590,Z 665.485,A 0.000,B 0.000,C 90.000,E1 267.364} C_DIS
LIN {X -0.020,Y -455.341,Z 665.484,A 0.000,B 0.000,C 90.000,E1 267.192} C_DIS
LIN {X 0.098,Y -448.262,Z 665.483,A 0.000,B 0.000,C 90.000,E1 266.846} C_DIS
LIN {X -0.175,Y -440.937,Z 665.481,A 0.000,B 0.000,C 90.000,E1 266.617} C_DIS
LIN {X 0.029,Y -432.741,Z 665.480,A 0.000,B 0.000,C 90.000,E1 266.388} C_DIS
LIN {X -0.179,Y -423.419,Z 665.479,A 0.000,B 0.000,C 90.000,E1 266.274} C_DIS
LIN {X -0.177,Y -414.862,Z 665.479,A 0.000,B 0.000,C 90.000,E1 266.216} C_DIS
LIN {X 0.080,Y -180.929,Z 665.479,A 0.000,B 0.000,C 90.000,E1 266.159} C_DIS
LIN {X -0.021,Y -180.904,Z 665.474,A 0.000,B 0.000,C 90.000,E1 265.298} C_DIS
LIN {X -0.071,Y -180.240,Z 665.464,A 0.000,B 0.000,C 90.000,E1 263.628} C_DIS
LIN {X -0.052,Y -178.727,Z 665.441,A 0.000,B 0.000,C 90.000,E1 259.398} C_DIS
LIN {X 0.015,Y -175.775,Z 665.413,A 0.000,B 0.000,C 90.000,E1 254.283} C_DIS
LIN {X 0.003,Y -171.958,Z 665.384,A 0.000,B 0.000,C 90.000,E1 249.156} C_DIS
LIN {X 0.041,Y -171.352,Z 665.379,A 0.000,B 0.000,C 90.000,E1 248.284} C_DIS
LIN {X 0.019,Y -167.603,Z 665.355,A 0.000,B 0.000,C 90.000,E1 243.973} C_DIS
LIN {X 0.031,Y -166.247,Z 665.346,A 0.000,B 0.000,C 90.000,E1 242.231} C_DIS
LIN {X 0.019,Y -163.003,Z 665.326,A 0.000,B 0.000,C 90.000,E1 238.742} C_DIS
LIN {X 0.065,Y -160.924,Z 665.312,A 0.000,B 0.000,C 90.000,E1 236.087} C_DIS
LIN {X 0.042,Y -157.686,Z 665.292,A 0.000,B 0.000,C 90.000,E1 232.557} C_DIS
LIN {X -0.019,Y -155.726,Z 665.277,A 0.000,B 0.000,C 90.000,E1 229.908} C_DIS
LIN {X 0.035,Y -151.985,Z 665.252,A 0.000,B 0.000,C 90.000,E1 225.405} C_DIS
LIN {X 0.051,Y -150.229,Z 665.237,A 0.000,B 0.000,C 90.000,E1 222.690} C_DIS
LIN {X -0.026,Y -146.990,Z 665.212,A 0.000,B 0.000,C 90.000,E1 218.177} C_DIS
LIN {X -0.035,Y -145.576,Z 665.197,A 0.000,B 0.000,C 90.000,E1 215.438} C_DIS
LIN {X 0.081,Y -142.965,Z 665.171,A 0.000,B 0.000,C 90.000,E1 210.797} C_DIS
LIN {X 0.012,Y -141.592,Z 665.151,A 0.000,B 0.000,C 90.000,E1 207.129} C_DIS
LIN {X 0.059,Y -139.421,Z 665.115,A 0.000,B 0.000,C 90.000,E1 200.610} C_DIS
LIN {X -0.021,Y -139.146,Z 665.104,A 0.000,B 0.000,C 90.000,E1 198.779} C_DIS
LIN {X 0.001,Y -138.346,Z 665.058,A 0.000,B 0.000,C 90.000,E1 190.366} C_DIS
LIN {X -0.013,Y -139.488,Z 665.006,A 0.000,B 0.000,C 90.000,E1 181.031} C_DIS
LIN {X 0.067,Y -141.092,Z 664.975,A 0.000,B 0.000,C 90.000,E1 175.412} C_DIS
LIN {X 0.021,Y -142.470,Z 664.959,A 0.000,B 0.000,C 90.000,E1 172.648} C_DIS
LIN {X -0.031,Y -144.716,Z 664.934,A 0.000,B 0.000,C 90.000,E1 168.049} C_DIS
LIN {X 0.062,Y -147.316,Z 664.913,A 0.000,B 0.000,C 90.000,E1 164.338} C_DIS
LIN {X -0.066,Y -150.637,Z 664.888,A 0.000,B 0.000,C 90.000,E1 159.826} C_DIS
LIN {X 0.010,Y -154.114,Z 664.868,A 0.000,B 0.000,C 90.000,E1 156.177} C_DIS
LIN {X -0.066,Y -157.539,Z 664.848,A 0.000,B 0.000,C 90.000,E1 152.615} C_DIS
LIN {X 0.100,Y -161.776,Z 664.828,A 0.000,B 0.000,C 90.000,E1 148.997} C_DIS
LIN {X -0.017,Y -165.969,Z 664.808,A 0.000,B 0.000,C 90.000,E1 145.515} C_DIS
LIN {X -0.021,Y -170.963,Z 664.789,A 0.000,B 0.000,C 90.000,E1 142.029} C_DIS
LIN {X 0.030,Y -175.832,Z 664.770,A 0.000,B 0.000,C 90.000,E1 138.566} C_DIS
LIN {X 0.025,Y -181.438,Z 664.751,A 0.000,B 0.000,C 90.000,E1 135.162} C_DIS
LIN {X -0.101,Y -186.944,Z 664.732,A 0.000,B 0.000,C 90.000,E1 131.838} C_DIS
LIN {X 0.105,Y -191.064,Z 664.720,A 0.000,B 0.000,C 90.000,E1 129.564} C_DIS
LIN {X 0.107,Y -288.653,Z 664.720,A 0.000,B 0.000,C 90.000,E1 129.564} C_DIS
LIN {X 0.053,Y -293.265,Z 664.719,A 0.000,B 0.000,C 90.000,E1 129.439} C_DIS
LIN {X -0.045,Y -295.383,Z 664.718,A 0.000,B 0.000,C 90.000,E1 129.322} C_DIS
LIN {X 0.068,Y -299.248,Z 664.716,A 0.000,B 0.000,C 90.000,E1 128.910} C_DIS
LIN {X 0.075,Y -302.741,Z 664.713,A 0.000,B 0.000,C 90.000,E1 128.338} C_DIS
LIN {X 0.025,Y -304.165,Z 664.711,A 0.000,B 0.000,C 90.000,E1 128.016} C_DIS
LIN {X 0.027,Y -305.284,Z 664.709,A 0.000,B 0.000,C 90.000,E1 127.684} C_DIS
LIN {X -0.103,Y -315.855,Z 664.689,A 0.000,B 0.000,C 90.000,E1 124.119} C_DIS
LIN {X 0.053,Y -325.844,Z 664.673,A 0.000,B 0.000,C 90.000,E1 121.209} C_DIS
LIN {X 0.176,Y -337.155,Z 664.658,A 0.000,B 0.000,C 90.000,E1 118.359} C_DIS
LIN {X 0.138,Y -349.893,Z 664.642,A 0.000,B 0.000,C 90.000,E1 115.591} C_DIS
LIN {X -0.052,Y -362.503,Z 664.629,A 0.000,B 0.000,C 90.000,E1 113.206} C_DIS
LIN {X -0.078,Y -376.419,Z 664.616,A 0.000,B 0.000,C 90.000,E1 110.844} C_DIS
LIN {X -0.161,Y -391.740,Z 664.603,A 0.000,B 0.000,C 90.000,E1 108.544} C_DIS
LIN {X 0.024,Y -408.580,Z 664.590,A 0.000,B 0.000,C 90.000,E1 106.260} C_DIS
LIN {X 0.009,Y -427.060,Z 664.578,A 0.000,B 0.000,C 90.000,E1 104.064} C_DIS
LIN {X 0.110,Y -446.947,Z 664.566,A 0.000,B 0.000,C 90.000,E1 101.951} C_DIS
LIN {X 0.127,Y -469.969,Z 664.555,A 0.000,B 0.000,C 90.000,E1 99.792} C_DIS
LIN {X 0.187,Y -471.988,Z 664.553,A 0.000,B 0.000,C 90.000,E1 99.557} C_DIS
LIN {X 0.041,Y -473.676,Z 664.552,A 0.000,B 0.000,C 90.000,E1 99.321} C_DIS
LIN {X -0.182,Y -474.943,Z 664.550,A 0.000,B 0.000,C 90.000,E1 99.095} C_DIS
LIN {X 0.012,Y -476.511,Z 664.548,A 0.000,B 0.000,C 90.000,E1 98.568} C_DIS
LIN {X 0.143,Y -477.027,Z 664.545,A 0.000,B 0.000,C 90.000,E1 98.049} C_DIS
LIN {X -0.190,Y -476.578,Z 664.542,A 0.000,B 0.000,C 90.000,E1 97.587} C_DIS
LIN {X -0.044,Y -475.096,Z 664.539,A 0.000,B 0.000,C 90.000,E1 97.068} C_DIS
LIN {X -0.179,Y -473.890,Z 664.538,A 0.000,B 0.000,C 90.000,E1 96.834} C_DIS
LIN {X 0.068,Y -467.067,Z 664.532,A 0.000,B 0.000,C 90.000,E1 95.796} C_DIS
LIN {X 0.045,Y -452.282,Z 664.519,A 0.000,B 0.000,C 90.000,E1 93.498} C_DIS
LIN {X -0.024,Y -436.194,Z 664.503,A 0.000,B 0.000,C 90.000,E1 90.630} C_DIS
LIN {X -0.108,Y -428.817,Z 664.496,A 0.000,B 0.000,C 90.000,E1 89.312} C_DIS
LIN {X -0.063,Y -417.983,Z 664.486,A 0.000,B 0.000,C 90.000,E1 87.421} C_DIS
LIN {X 0.191,Y -407.098,Z 664.475,A 0.000,B 0.000,C 90.000,E1 85.469} C_DIS
LIN {X -0.067,Y -393.284,Z 664.461,A 0.000,B 0.000,C 90.000,E1 82.996} C_DIS
LIN {X -0.138,Y -379.930,Z 664.447,A 0.000,B 0.000,C 90.000,E1 80.443} C_DIS
LIN {X -0.117,Y -368.505,Z 664.434,A 0.000,B 0.000,C 90.000,E1 78.117} C_DIS
LIN {X 0.159,Y -356.033,Z 664.419,A 0.000,B 0.000,C 90.000,E1 75.408} C_DIS
LIN {X 0.025,Y -345.546,Z 664.406,A 0.000,B 0.000,C 90.000,E1 73.015} C_DIS
LIN {X 0.037,Y -331.839,Z 664.387,A 0.000,B 0.000,C 90.000,E1 69.625} C_DIS
LIN {X -0.066,Y -319.252,Z 664.368,A 0.000,B 0.000,C 90.000,E1 66.177} C_DIS
LIN {X 0.081,Y -308.023,Z 664.348,A 0.000,B 0.000,C 90.000,E1 62.615} C_DIS
LIN {X 0.139,Y -298.798,Z 664.330,A 0.000,B 0.000,C 90.000,E1 59.331} C_DIS
LIN {X -0.032,Y -292.009,Z 664.315,A 0.000,B 0.000,C 90.000,E1 56.707} C_DIS
LIN {X 0.108,Y -285.467,Z 664.300,A 0.000,B 0.000,C 90.000,E1 53.989} C_DIS
LIN {X -0.058,Y -280.596,Z 664.289,A 0.000,B 0.000,C 90.000,E1 51.984} C_DIS
LIN {X 0.033,Y -275.441,Z 664.277,A 0.000,B 0.000,C 90.000,E1 49.908} C_DIS
LIN {X -0.001,Y -269.971,Z 664.266,A 0.000,B 0.000,C 90.000,E1 47.838} C_DIS
LIN {X 0.044,Y -264.085,Z 664.254,A 0.000,B 0.000,C 90.000,E1 45.729} C_DIS
LIN {X -0.030,Y -257.864,Z 664.242,A 0.000,B 0.000,C 90.000,E1 43.623} C_DIS
LIN {X -0.020,Y -251.381,Z 664.230,A 0.000,B 0.000,C 90.000,E1 41.472} C_DIS
LIN {X 0.068,Y -242.782,Z 664.214,A 0.000,B 0.000,C 90.000,E1 38.543} C_DIS
LIN {X 0.016,Y -234.708,Z 664.198,A 0.000,B 0.000,C 90.000,E1 35.598} C_DIS
LIN {X -0.119,Y -227.282,Z 664.181,A 0.000,B 0.000,C 90.000,E1 32.625} C_DIS
LIN {X 0.015,Y -220.566,Z 664.164,A 0.000,B 0.000,C 90.000,E1 29.539} C_DIS
LIN {X 0.040,Y -214.673,Z 664.147,A 0.000,B 0.000,C 90.000,E1 26.437} C_DIS
LIN {X -0.071,Y -209.642,Z 664.130,A 0.000,B 0.000,C 90.000,E1 23.334} C_DIS
LIN {X 0.104,Y -204.397,Z 664.107,A 0.000,B 0.000,C 90.000,E1 19.322} C_DIS
LIN {X -0.089,Y -200.269,Z 664.085,A 0.000,B 0.000,C 90.000,E1 15.371} C_DIS
LIN {X 0.013,Y -196.696,Z 664.058,A 0.000,B 0.000,C 90.000,E1 10.489} C_DIS
LIN {X 0.056,Y -194.166,Z 664.022,A 0.000,B 0.000,C 90.000,E1 3.955} C_DIS
LIN {X -0.023,Y -195.719,Z 663.961,A 0.000,B 0.000,C 90.000,E1 352.996} C_DIS
LIN {X -0.043,Y -198.744,Z 663.934,A 0.000,B 0.000,C 90.000,E1 348.117} C_DIS
LIN {X 0.055,Y -202.403,Z 663.911,A 0.000,B 0.000,C 90.000,E1 344.047} C_DIS
LIN {X -0.024,Y -207.058,Z 663.889,A 0.000,B 0.000,C 90.000,E1 340.061} C_DIS
LIN {X -0.052,Y -212.489,Z 663.867,A 0.000,B 0.000,C 90.000,E1 336.102} C_DIS
LIN {X 0.057,Y -218.702,Z 663.845,A 0.000,B 0.000,C 90.000,E1 332.153} C_DIS
LIN {X -0.106,Y -225.578,Z 663.824,A 0.000,B 0.000,C 90.000,E1 328.329} C_DIS
LIN {X -0.052,Y -231.517,Z 663.807,A 0.000,B 0.000,C 90.000,E1 325.261} C_DIS
LIN {X 0.120,Y -239.445,Z 663.786,A 0.000,B 0.000,C 90.000,E1 321.457} C_DIS
LIN {X -0.054,Y -248.176,Z 663.765,A 0.000,B 0.000,C 90.000,E1 317.796} C_DIS
LIN {X -0.007,Y -257.916,Z 663.745,A 0.000,B 0.000,C 90.000,E1 314.150} C_DIS
LIN {X -0.010,Y -267.715,Z 663.727,A 0.000,B 0.000,C 90.000,E1 310.943} C_DIS
LIN {X -0.064,Y -278.731,Z 663.710,A 0.000,B 0.000,C 90.000,E1 307.810} C_DIS
LIN {X -0.123,Y -292.213,Z 663.691,A 0.000,B 0.000,C 90.000,E1 304.405} C_DIS
LIN {X 0.001,Y -307.361,Z 663.672,A 0.000,B 0.000,C 90.000,E1 301.052} C_DIS
LIN {X -0.179,Y -323.891,Z 663.655,A 0.000,B 0.000,C 90.000,E1 297.847} C_DIS
LIN {X 0.079,Y -336.123,Z 663.642,A 0.000,B 0.000,C 90.000,E1 295.591} C_DIS
LIN {X 0.077,Y -354.309,Z 663.625,A 0.000,B 0.000,C 90.000,E1 292.514} C_DIS
LIN {X 0.069,Y -369.758,Z 663.612,A 0.000,B 0.000,C 90.000,E1 290.120} C_DIS
LIN {X 0.075,Y -382.618,Z 663.602,A 0.000,B 0.000,C 90.000,E1 288.362} C_DIS
LIN {X 0.118,Y -403.429,Z 663.588,A 0.000,B 0.000,C 90.000,E1 285.788} C_DIS
LIN {X 0.017,Y -415.013,Z 663.580,A 0.000,B 0.000,C 90.000,E1 284.411} C_DIS
LIN {X -0.133,Y -426.161,Z 663.572,A 0.000,B 0.000,C 90.000,E1 283.063} C_DIS
LIN {X 0.128,Y -434.646,Z 663.566,A 0.000,B 0.000,C 90.000,E1 281.951} C_DIS
LIN {X -0.151,Y -444.676,Z 663.559,A 0.000,B 0.000,C 90.000,E1 280.658} C_DIS
LIN {X 0.055,Y -458.757,Z 663.549,A 0.000,B 0.000,C 90.000,E1 278.803} C_DIS
LIN {X -0.094,Y -465.129,Z 663.545,A 0.000,B 0.000,C 90.000,E1 278.049} C_DIS
LIN {X -0.199,Y -470.881,Z 663.540,A 0.000,B 0.000,C 90.000,E1 277.296} C_DIS
LIN {X -0.103,Y -474.203,Z 663.538,A 0.000,B 0.000,C 90.000,E1 276.777} C_DIS
LIN {X 0.015,Y -477.152,Z 663.535,A 0.000,B 0.000,C 90.000,E1 276.258} C_DIS
LIN {X -0.032,Y -480.853,Z 663.531,A 0.000,B 0.000,C 90.000,E1 275.511} C_DIS
LIN {X -0.172,Y -481.932,Z 663.529,A 0.000,B 0.000,C 90.000,E1 275.277} C_DIS
LIN {X -0.007,Y -483.777,Z 663.526,A 0.000,B 0.000,C 90.000,E1 274.759} C_DIS
LIN {X 0.128,Y -485.175,Z 663.524,A 0.000,B 0.000,C 90.000,E1 274.245} C_DIS
LIN {X -0.174,Y -486.172,Z 663.521,A 0.000,B 0.000,C 90.000,E1 273.784} C_DIS
LIN {X -0.015,Y -486.813,Z 663.518,A 0.000,B 0.000,C 90.000,E1 273.269} C_DIS
LIN {X 0.179,Y -487.163,Z 663.515,A 0.000,B 0.000,C 90.000,E1 272.751} C_DIS
LIN {X -0.135,Y -487.205,Z 663.513,A 0.000,B 0.000,C 90.000,E1 272.293} C_DIS
LIN {X 0.058,Y -486.892,Z 663.510,A 0.000,B 0.000,C 90.000,E1 271.776} C_DIS
LIN {X 0.233,Y -486.256,Z 663.507,A 0.000,B 0.000,C 90.000,E1 271.260} C_DIS
LIN {X -0.078,Y -485.238,Z 663.504,A 0.000,B 0.000,C 90.000,E1 270.802} C_DIS
LIN {X 0.095,Y -483.736,Z 663.502,A 0.000,B 0.000,C 90.000,E1 270.286} C_DIS
LIN {X -0.221,Y -481.684,Z 663.499,A 0.000,B 0.000,C 90.000,E1 269.828} C_DIS
LIN {X -0.064,Y -478.897,Z 663.496,A 0.000,B 0.000,C 90.000,E1 269.312} C_DIS
LIN {X 0.073,Y -475.339,Z 663.493,A 0.000,B 0.000,C 90.000,E1 268.797} C_DIS
LIN {X 0.187,Y -470.704,Z 663.491,A 0.000,B 0.000,C 90.000,E1 268.282} C_DIS
LIN {X 0.031,Y -468.007,Z 663.489,A 0.000,B 0.000,C 90.000,E1 268.051} C_DIS
LIN {X -0.026,Y -462.019,Z 663.487,A 0.000,B 0.000,C 90.000,E1 267.593} C_DIS
LIN {X 0.004,Y -455.465,Z 663.484,A 0.000,B 0.000,C 90.000,E1 267.192} C_DIS
LIN {X 0.121,Y -448.515,Z 663.483,A 0.000,B 0.000,C 90.000,E1 266.849} C_DIS
LIN {X -0.119,Y -441.208,Z 663.481,A 0.000,B 0.000,C 90.000,E1 266.617} C_DIS
LIN {X 0.082,Y -433.229,Z 663.480,A 0.000,B 0.000,C 90.000,E1 266.388} C_DIS
LIN {X -0.151,Y -424.117,Z 663.479,A 0.000,B 0.000,C 90.000,E1 266.274} C_DIS
LIN {X 0.194,Y -414.536,Z 663.479,A 0.000,B 0.000,C 90.000,E1 266.159} C_DIS
LIN {X 0.059,Y -180.928,Z 663.479,A 0.000,B 0.000,C 90.000,E1 266.159} C_DIS
LIN {X -0.032,Y -180.903,Z 663.474,A 0.000,B 0.000,C 90.000,E1 265.298} C_DIS
LIN {X -0.082,Y -180.238,Z 663.464,A 0.000,B 0.000,C 90.000,E1 263.628} C_DIS
LIN {X -0.063,Y -178.725,Z 663.441,A 0.000,B 0.000,C 90.000,E1 259.398} C_DIS
LIN {X 0.004,Y -175.773,Z 663.413,A 0.000,B 0.000,C 90.000,E1 254.283} C_DIS
LIN {X -0.007,Y -171.957,Z 663.384,A 0.000,B 0.000,C 90.000,E1 249.156} C_DIS
LIN {X 0.030,Y -171.349,Z 663.379,A 0.000,B 0.000,C 90.000,E1 248.284} C_DIS
LIN {X 0.009,Y -167.600,Z 663.355,A 0.000,B 0.000,C 90.000,E1 243.973} C_DIS
LIN {X 0.021,Y -166.242,Z 663.346,A 0.000,B 0.000,C 90.000,E1 242.231} C_DIS
LIN {X 0.008,Y -163.001,Z 663.326,A 0.000,B 0.000,C 90.000,E1 238.742} C_DIS
LIN {X 0.055,Y -160.920,Z 663.312,A 0.000,B 0.000,C 90.000,E1 236.087} C_DIS
LIN {X 0.032,Y -157.683,Z 663.292,A 0.000,B 0.000,C 90.000,E1 232.557} C_DIS
LIN {X -0.029,Y -155.722,Z 663.277,A 0.000,B 0.000,C 90.000,E1 229.908} C_DIS
LIN {X 0.025,Y -151.982,Z 663.252,A 0.000,B 0.000,C 90.000,E1 225.405} C_DIS
LIN {X 0.041,Y -150.226,Z 663.237,A 0.000,B 0.000,C 90.000,E1 222.690} C_DIS
LIN {X -0.036,Y -146.988,Z 663.212,A 0.000,B 0.000,C 90.000,E1 218.177} C_DIS
LIN {X -0.046,Y -145.574,Z 663.197,A 0.000,B 0.000,C 90.000,E1 215.438} C_DIS
LIN {X 0.071,Y -142.964,Z 663.171,A 0.000,B 0.000,C 90.000,E1 210.797} C_DIS
LIN {X 0.002,Y -141.590,Z 663.151,A 0.000,B 0.000,C 90.000,E1 207.129} C_DIS
LIN {X 0.050,Y -139.419,Z 663.115,A 0.000,B 0.000,C 90.000,E1 200.610} C_DIS
LIN {X -0.030,Y -139.145,Z 663.104,A 0.000,B 0.000,C 90.000,E1 198.779} C_DIS
LIN {X -0.008,Y -138.347,Z 663.058,A 0.000,B 0.000,C 90.000,E1 190.366} C_DIS
LIN {X -0.023,Y -139.488,Z 663.006,A 0.000,B 0.000,C 90.000,E1 181.031} C_DIS
LIN {X 0.057,Y -141.093,Z 662.975,A 0.000,B 0.000,C 90.000,E1 175.412} C_DIS
LIN {X 0.011,Y -142.472,Z 662.959,A 0.000,B 0.000,C 90.000,E1 172.648} C_DIS
LIN {X -0.040,Y -144.718,Z 662.934,A 0.000,B 0.000,C 90.000,E1 168.049} C_DIS
LIN {X 0.053,Y -147.319,Z 662.913,A 0.000,B 0.000,C 90.000,E1 164.338} C_DIS
LIN {X -0.023,Y -150.640,Z 662.888,A 0.000,B 0.000,C 90.000,E1 159.806} C_DIS
LIN {X 0.000,Y -154.117,Z 662.868,A 0.000,B 0.000,C 90.000,E1 156.177} C_DIS
LIN {X -0.076,Y -157.543,Z 662.848,A 0.000,B 0.000,C 90.000,E1 152.615} C_DIS
LIN {X 0.089,Y -161.781,Z 662.828,A 0.000,B 0.000,C 90.000,E1 148.997} C_DIS
LIN {X -0.028,Y -165.973,Z 662.808,A 0.000,B 0.000,C 90.000,E1 145.515} C_DIS
LIN {X -0.032,Y -170.968,Z 662.789,A 0.000,B 0.000,C 90.000,E1 142.029} C_DIS
LIN {X 0.020,Y -175.837,Z 662.770,A 0.000,B 0.000,C 90.000,E1 138.566} C_DIS
LIN {X 0.014,Y -181.444,Z 662.751,A 0.000,B 0.000,C 90.000,E1 135.162} C_DIS
LIN {X -0.112,Y -186.951,Z 662.732,A 0.000,B 0.000,C 90.000,E1 131.838} C_DIS
LIN {X 0.008,Y -191.052,Z 662.720,A 0.000,B 0.000,C 90.000,E1 129.600} C_DIS
LIN {X 0.143,Y -288.402,Z 662.720,A 0.000,B 0.000,C 90.000,E1 129.564} C_DIS
LIN {X 0.091,Y -289.461,Z 662.720,A 0.000,B 0.000,C 90.000,E1 129.564} C_DIS
LIN {X -0.062,Y -295.467,Z 662.718,A 0.000,B 0.000,C 90.000,E1 129.322} C_DIS
LIN {X -0.042,Y -298.407,Z 662.717,A 0.000,B 0.000,C 90.000,E1 129.036} C_DIS
LIN {X 0.078,Y -302.097,Z 662.714,A 0.000,B 0.000,C 90.000,E1 128.463} C_DIS
LIN {X -0.162,Y -303.653,Z 662.712,A 0.000,B 0.000,C 90.000,E1 128.177} C_DIS
LIN {X 0.023,Y -304.877,Z 662.710,A 0.000,B 0.000,C 90.000,E1 127.810} C_DIS
LIN {X -0.070,Y -316.484,Z 662.688,A 0.000,B 0.000,C 90.000,E1 123.913} C_DIS
LIN {X 0.107,Y -326.558,Z 662.672,A 0.000,B 0.000,C 90.000,E1 121.003} C_DIS
LIN {X 0.087,Y -337.967,Z 662.657,A 0.000,B 0.000,C 90.000,E1 118.180} C_DIS
LIN {X 0.081,Y -350.803,Z 662.641,A 0.000,B 0.000,C 90.000,E1 115.412} C_DIS
LIN {X -0.081,Y -363.511,Z 662.628,A 0.000,B 0.000,C 90.000,E1 113.025} C_DIS
LIN {X -0.081,Y -377.531,Z 662.615,A 0.000,B 0.000,C 90.000,E1 110.663} C_DIS
LIN {X -0.135,Y -392.966,Z 662.602,A 0.000,B 0.000,C 90.000,E1 108.362} C_DIS
LIN {X 0.082,Y -409.928,Z 662.589,A 0.000,B 0.000,C 90.000,E1 106.079} C_DIS
LIN {X 0.102,Y -428.542,Z 662.577,A 0.000,B 0.000,C 90.000,E1 103.883} C_DIS
LIN {X -0.134,Y -448.481,Z 662.566,A 0.000,B 0.000,C 90.000,E1 101.827} C_DIS
LIN {X -0.093,Y -469.008,Z 662.555,A 0.000,B 0.000,C 90.000,E1 99.905} C_DIS
LIN {X -0.042,Y -471.299,Z 662.554,A 0.000,B 0.000,C 90.000,E1 99.670} C_DIS
LIN {X -0.142,Y -473.144,Z 662.552,A 0.000,B 0.000,C 90.000,E1 99.434} C_DIS
LIN {X 0.149,Y -474.538,Z 662.551,A 0.000,B 0.000,C 90.000,E1 99.151} C_DIS
LIN {X -0.129,Y -476.357,Z 662.548,A 0.000,B 0.000,C 90.000,E1 98.681} C_DIS
LIN {X -0.004,Y -477.084,Z 662.545,A 0.000,B 0.000,C 90.000,E1 98.163} C_DIS
LIN {X 0.136,Y -476.837,Z 662.543,A 0.000,B 0.000,C 90.000,E1 97.644} C_DIS
LIN {X -0.193,Y -475.586,Z 662.540,A 0.000,B 0.000,C 90.000,E1 97.182} C_DIS
LIN {X 0.143,Y -474.524,Z 662.538,A 0.000,B 0.000,C 90.000,E1 96.891} C_DIS
LIN {X -0.048,Y -473.100,Z 662.537,A 0.000,B 0.000,C 90.000,E1 96.663} C_DIS
LIN {X -0.103,Y -456.155,Z 662.523,A 0.000,B 0.000,C 90.000,E1 94.131} C_DIS
LIN {X -0.156,Y -444.011,Z 662.511,A 0.000,B 0.000,C 90.000,E1 92.064} C_DIS
LIN {X 0.049,Y -435.388,Z 662.503,A 0.000,B 0.000,C 90.000,E1 90.458} C_DIS
LIN {X -0.052,Y -427.994,Z 662.495,A 0.000,B 0.000,C 90.000,E1 89.141} C_DIS
LIN {X -0.022,Y -417.160,Z 662.485,A 0.000,B 0.000,C 90.000,E1 87.249} C_DIS
LIN {X -0.198,Y -406.243,Z 662.474,A 0.000,B 0.000,C 90.000,E1 85.355} C_DIS
LIN {X -0.027,Y -392.463,Z 662.460,A 0.000,B 0.000,C 90.000,E1 82.818} C_DIS
LIN {X -0.177,Y -379.156,Z 662.446,A 0.000,B 0.000,C 90.000,E1 80.274} C_DIS
LIN {X -0.106,Y -367.767,Z 662.433,A 0.000,B 0.000,C 90.000,E1 77.937} C_DIS
LIN {X 0.105,Y -354.046,Z 662.416,A 0.000,B 0.000,C 90.000,E1 74.936} C_DIS
LIN {X -0.077,Y -343.650,Z 662.403,A 0.000,B 0.000,C 90.000,E1 72.543} C_DIS
LIN {X -0.043,Y -328.972,Z 662.382,A 0.000,B 0.000,C 90.000,E1 68.827} C_DIS
LIN {X -0.111,Y -316.677,Z 662.363,A 0.000,B 0.000,C 90.000,E1 65.357} C_DIS
LIN {X 0.140,Y -304.833,Z 662.341,A 0.000,B 0.000,C 90.000,E1 61.435} C_DIS
LIN {X 0.020,Y -294.245,Z 662.319,A 0.000,B 0.000,C 90.000,E1 57.502} C_DIS
LIN {X 0.060,Y -287.661,Z 662.305,A 0.000,B 0.000,C 90.000,E1 54.815} C_DIS
LIN {X 0.030,Y -281.155,Z 662.290,A 0.000,B 0.000,C 90.000,E1 52.110} C_DIS
LIN {X -0.043,Y -276.064,Z 662.278,A 0.000,B 0.000,C 90.000,E1 50.070} C_DIS
LIN {X -0.066,Y -270.605,Z 662.267,A 0.000,B 0.000,C 90.000,E1 48.000} C_DIS
LIN {X -0.008,Y -264.759,Z 662.255,A 0.000,B 0.000,C 90.000,E1 45.891} C_DIS
LIN {X -0.069,Y -258.521,Z 662.243,A 0.000,B 0.000,C 90.000,E1 43.785} C_DIS
LIN {X 0.123,Y -252.045,Z 662.231,A 0.000,B 0.000,C 90.000,E1 41.595} C_DIS
LIN {X -0.127,Y -243.412,Z 662.215,A 0.000,B 0.000,C 90.000,E1 38.749} C_DIS
LIN {X 0.031,Y -235.310,Z 662.199,A 0.000,B 0.000,C 90.000,E1 35.758} C_DIS
LIN {X 0.039,Y -227.844,Z 662.182,A 0.000,B 0.000,C 90.000,E1 32.752} C_DIS
LIN {X -0.011,Y -221.075,Z 662.165,A 0.000,B 0.000,C 90.000,E1 29.716} C_DIS
LIN {X 0.021,Y -215.142,Z 662.148,A 0.000,B 0.000,C 90.000,E1 26.616} C_DIS
LIN {X -0.083,Y -210.066,Z 662.130,A 0.000,B 0.000,C 90.000,E1 23.515} C_DIS
LIN {X 0.035,Y -204.762,Z 662.109,A 0.000,B 0.000,C 90.000,E1 19.523} C_DIS
LIN {X -0.079,Y -200.573,Z 662.086,A 0.000,B 0.000,C 90.000,E1 15.552} C_DIS
LIN {X 0.074,Y -196.922,Z 662.059,A 0.000,B 0.000,C 90.000,E1 10.658} C_DIS
LIN {X -0.090,Y -194.302,Z 662.023,A 0.000,B 0.000,C 90.000,E1 4.188} C_DIS
LIN {X -0.019,Y -195.801,Z 661.961,A 0.000,B 0.000,C 90.000,E1 352.996} C_DIS
LIN {X -0.034,Y -198.832,Z 661.934,A 0.000,B 0.000,C 90.000,E1 348.117} C_DIS
LIN {X 0.066,Y -202.471,Z 661.911,A 0.000,B 0.000,C 90.000,E1 344.047} C_DIS
LIN {X -0.012,Y -207.113,Z 661.889,A 0.000,B 0.000,C 90.000,E1 340.061} C_DIS
LIN {X -0.037,Y -212.540,Z 661.867,A 0.000,B 0.000,C 90.000,E1 336.102} C_DIS
LIN {X 0.074,Y -218.761,Z 661.845,A 0.000,B 0.000,C 90.000,E1 332.153} C_DIS
LIN {X -0.088,Y -225.638,Z 661.824,A 0.000,B 0.000,C 90.000,E1 328.329} C_DIS
LIN {X 0.058,Y -233.094,Z 661.803,A 0.000,B 0.000,C 90.000,E1 324.482} C_DIS
LIN {X 0.095,Y -241.164,Z 661.782,A 0.000,B 0.000,C 90.000,E1 320.723} C_DIS
LIN {X -0.047,Y -250.036,Z 661.761,A 0.000,B 0.000,C 90.000,E1 317.067} C_DIS
LIN {X -0.117,Y -259.982,Z 661.741,A 0.000,B 0.000,C 90.000,E1 313.461} C_DIS
LIN {X -0.050,Y -270.007,Z 661.724,A 0.000,B 0.000,C 90.000,E1 310.253} C_DIS
LIN {X -0.103,Y -282.602,Z 661.704,A 0.000,B 0.000,C 90.000,E1 306.790} C_DIS
LIN {X 0.037,Y -295.052,Z 661.687,A 0.000,B 0.000,C 90.000,E1 303.706} C_DIS
LIN {X -0.062,Y -310.462,Z 661.669,A 0.000,B 0.000,C 90.000,E1 300.413} C_DIS
LIN {X 0.017,Y -327.289,Z 661.651,A 0.000,B 0.000,C 90.000,E1 297.180} C_DIS
LIN {X 0.061,Y -339.552,Z 661.639,A 0.000,B 0.000,C 90.000,E1 294.975} C_DIS
LIN {X 0.131,Y -356.111,Z 661.623,A 0.000,B 0.000,C 90.000,E1 292.206} C_DIS
LIN {X 0.089,Y -369.651,Z 661.612,A 0.000,B 0.000,C 90.000,E1 290.120} C_DIS
LIN {X 0.093,Y -382.508,Z 661.602,A 0.000,B 0.000,C 90.000,E1 288.362} C_DIS
LIN {X 0.135,Y -403.320,Z 661.588,A 0.000,B 0.000,C 90.000,E1 285.788} C_DIS
LIN {X 0.032,Y -414.904,Z 661.580,A 0.000,B 0.000,C 90.000,E1 284.411} C_DIS
LIN {X -0.119,Y -426.054,Z 661.573,A 0.000,B 0.000,C 90.000,E1 283.063} C_DIS
LIN {X -0.095,Y -436.575,Z 661.565,A 0.000,B 0.000,C 90.000,E1 281.715} C_DIS
LIN {X 0.079,Y -446.530,Z 661.558,A 0.000,B 0.000,C 90.000,E1 280.366} C_DIS
LIN {X -0.195,Y -456.569,Z 661.550,A 0.000,B 0.000,C 90.000,E1 279.095} C_DIS
LIN {X -0.085,Y -465.106,Z 661.545,A 0.000,B 0.000,C 90.000,E1 278.049} C_DIS
LIN {X -0.191,Y -470.891,Z 661.540,A 0.000,B 0.000,C 90.000,E1 277.296} C_DIS
LIN {X 0.228,Y -475.727,Z 661.536,A 0.000,B 0.000,C 90.000,E1 276.486} C_DIS
LIN {X 0.162,Y -479.704,Z 661.532,A 0.000,B 0.000,C 90.000,E1 275.739} C_DIS
LIN {X -0.163,Y -481.918,Z 661.529,A 0.000,B 0.000,C 90.000,E1 275.277} C_DIS
LIN {X 0.002,Y -483.734,Z 661.526,A 0.000,B 0.000,C 90.000,E1 274.759} C_DIS
LIN {X 0.136,Y -485.152,Z 661.524,A 0.000,B 0.000,C 90.000,E1 274.245} C_DIS
LIN {X -0.166,Y -486.123,Z 661.521,A 0.000,B 0.000,C 90.000,E1 273.784} C_DIS
LIN {X -0.007,Y -486.792,Z 661.518,A 0.000,B 0.000,C 90.000,E1 273.269} C_DIS
LIN {X 0.186,Y -487.112,Z 661.515,A 0.000,B 0.000,C 90.000,E1 272.751} C_DIS
LIN {X -0.128,Y -487.158,Z 661.513,A 0.000,B 0.000,C 90.000,E1 272.293} C_DIS
LIN {X 0.064,Y -486.876,Z 661.510,A 0.000,B 0.000,C 90.000,E1 271.776} C_DIS
LIN {X 0.240,Y -486.245,Z 661.507,A 0.000,B 0.000,C 90.000,E1 271.260} C_DIS
LIN {X -0.070,Y -485.224,Z 661.504,A 0.000,B 0.000,C 90.000,E1 270.802} C_DIS
LIN {X 0.101,Y -483.733,Z 661.502,A 0.000,B 0.000,C 90.000,E1 270.286} C_DIS
LIN {X -0.215,Y -481.682,Z 661.499,A 0.000,B 0.000,C 90.000,E1 269.828} C_DIS
LIN {X -0.056,Y -478.914,Z 661.496,A 0.000,B 0.000,C 90.000,E1 269.312} C_DIS
LIN {X 0.079,Y -475.351,Z 661.493,A 0.000,B 0.000,C 90.000,E1 268.797} C_DIS
LIN {X 0.194,Y -470.759,Z 661.491,A 0.000,B 0.000,C 90.000,E1 268.282} C_DIS
LIN {X -0.155,Y -464.929,Z 661.488,A 0.000,B 0.000,C 90.000,E1 267.822} C_DIS
LIN {X -0.067,Y -462.021,Z 661.487,A 0.000,B 0.000,C 90.000,E1 267.593} C_DIS
LIN {X -0.041,Y -455.440,Z 661.484,A 0.000,B 0.000,C 90.000,E1 267.192} C_DIS
LIN {X 0.112,Y -448.470,Z 661.483,A 0.000,B 0.000,C 90.000,E1 266.846} C_DIS
LIN {X -0.171,Y -441.021,Z 661.481,A 0.000,B 0.000,C 90.000,E1 266.617} C_DIS
LIN {X 0.023,Y -433.125,Z 661.480,A 0.000,B 0.000,C 90.000,E1 266.388} C_DIS
LIN {X -0.194,Y -423.919,Z 661.479,A 0.000,B 0.000,C 90.000,E1 266.274} C_DIS
LIN {X 0.160,Y -414.587,Z 661.479,A 0.000,B 0.000,C 90.000,E1 266.159} C_DIS
LIN {X 0.045,Y -180.928,Z 661.479,A 0.000,B 0.000,C 90.000,E1 266.159} C_DIS
LIN {X -0.047,Y -180.903,Z 661.474,A 0.000,B 0.000,C 90.000,E1 265.298} C_DIS
LIN {X 0.083,Y -180.237,Z 661.464,A 0.000,B 0.000,C 90.000,E1 263.571} C_DIS
LIN {X -0.077,Y -178.722,Z 661.441,A 0.000,B 0.000,C 90.000,E1 259.398} C_DIS
LIN {X -0.009,Y -175.770,Z 661.413,A 0.000,B 0.000,C 90.000,E1 254.283} C_DIS
LIN {X -0.021,Y -171.954,Z 661.384,A 0.000,B 0.000,C 90.000,E1 249.156} C_DIS
LIN {X 0.017,Y -171.345,Z 661.379,A 0.000,B 0.000,C 90.000,E1 248.284} C_DIS
LIN {X -0.005,Y -167.597,Z 661.355,A 0.000,B 0.000,C 90.000,E1 243.973} C_DIS
LIN {X 0.007,Y -166.238,Z 661.346,A 0.000,B 0.000,C 90.000,E1 242.231} C_DIS
LIN {X -0.005,Y -162.996,Z 661.326,A 0.000,B 0.000,C 90.000,E1 238.742} C_DIS
LIN {X 0.042,Y -160.916,Z 661.312,A 0.000,B 0.000,C 90.000,E1 236.087} C_DIS
LIN {X 0.019,Y -157.679,Z 661.292,A 0.000,B 0.000,C 90.000,E1 232.557} C_DIS
LIN {X -0.043,Y -155.718,Z 661.277,A 0.000,B 0.000,C 90.000,E1 229.908} C_DIS
LIN {X 0.012,Y -151.979,Z 661.252,A 0.000,B 0.000,C 90.000,E1 225.405} C_DIS
LIN {X 0.028,Y -150.222,Z 661.237,A 0.000,B 0.000,C 90.000,E1 222.690} C_DIS
LIN {X -0.048,Y -146.986,Z 661.212,A 0.000,B 0.000,C 90.000,E1 218.177} C_DIS
LIN {X 0.061,Y -145.571,Z 661.197,A 0.000,B 0.000,C 90.000,E1 215.391} C_DIS
LIN {X 0.059,Y -142.961,Z 661.171,A 0.000,B 0.000,C 90.000,E1 210.797} C_DIS
LIN {X -0.010,Y -141.587,Z 661.151,A 0.000,B 0.000,C 90.000,E1 207.129} C_DIS
LIN {X 0.037,Y -139.419,Z 661.115,A 0.000,B 0.000,C 90.000,E1 200.610} C_DIS
LIN {X -0.043,Y -139.144,Z 661.104,A 0.000,B 0.000,C 90.000,E1 198.779} C_DIS
LIN {X -0.021,Y -138.346,Z 661.058,A 0.000,B 0.000,C 90.000,E1 190.366} C_DIS
LIN {X -0.035,Y -139.489,Z 661.006,A 0.000,B 0.000,C 90.000,E1 181.031} C_DIS
LIN {X 0.045,Y -141.095,Z 660.975,A 0.000,B 0.000,C 90.000,E1 175.412} C_DIS
LIN {X 0.000,Y -142.473,Z 660.959,A 0.000,B 0.000,C 90.000,E1 172.648} C_DIS
LIN {X -0.053,Y -144.721,Z 660.933,A 0.000,B 0.000,C 90.000,E1 168.049} C_DIS
LIN {X 0.039,Y -147.322,Z 660.913,A 0.000,B 0.000,C 90.000,E1 164.338} C_DIS
LIN {X -0.036,Y -150.645,Z 660.888,A 0.000,B 0.000,C 90.000,E1 159.806} C_DIS
LIN {X -0.013,Y -154.122,Z 660.868,A 0.000,B 0.000,C 90.000,E1 156.177} C_DIS
LIN {X -0.089,Y -157.548,Z 660.848,A 0.000,B 0.000,C 90.000,E1 152.615} C_DIS
LIN {X 0.076,Y -161.787,Z 660.828,A 0.000,B 0.000,C 90.000,E1 148.997} C_DIS
LIN {X -0.042,Y -165.979,Z 660.808,A 0.000,B 0.000,C 90.000,E1 145.515} C_DIS
LIN {X -0.046,Y -170.975,Z 660.789,A 0.000,B 0.000,C 90.000,E1 142.029} C_DIS
LIN {X 0.005,Y -175.845,Z 660.770,A 0.000,B 0.000,C 90.000,E1 138.566} C_DIS
LIN {X -0.001,Y -181.451,Z 660.751,A 0.000,B 0.000,C 90.000,E1 135.162} C_DIS
LIN {X -0.127,Y -186.959,Z 660.732,A 0.000,B 0.000,C 90.000,E1 131.838} C_DIS
LIN {X 0.115,Y -191.060,Z 660.720,A 0.000,B 0.000,C 90.000,E1 129.564} C_DIS
LIN {X 0.122,Y -289.275,Z 660.720,A 0.000,B 0.000,C 90.000,E1 129.564} C_DIS
LIN {X 0.144,Y -295.548,Z 660.718,A 0.000,B 0.000,C 90.000,E1 129.277} C_DIS
LIN {X 0.076,Y -298.598,Z 660.717,A 0.000,B 0.000,C 90.000,E1 128.991} C_DIS
LIN {X -0.091,Y -302.255,Z 660.714,A 0.000,B 0.000,C 90.000,E1 128.463} C_DIS
LIN {X 0.095,Y -303.769,Z 660.712,A 0.000,B 0.000,C 90.000,E1 128.096} C_DIS
LIN {X -0.146,Y -304.961,Z 660.710,A 0.000,B 0.000,C 90.000,E1 127.810} C_DIS
LIN {X -0.039,Y -315.520,Z 660.690,A 0.000,B 0.000,C 90.000,E1 124.199} C_DIS
LIN {X -0.165,Y -325.469,Z 660.674,A 0.000,B 0.000,C 90.000,E1 121.337} C_DIS
LIN {X -0.062,Y -336.737,Z 660.658,A 0.000,B 0.000,C 90.000,E1 118.487} C_DIS
LIN {X -0.122,Y -349.427,Z 660.643,A 0.000,B 0.000,C 90.000,E1 115.720} C_DIS
LIN {X 0.145,Y -361.992,Z 660.629,A 0.000,B 0.000,C 90.000,E1 113.259} C_DIS
LIN {X -0.027,Y -375.860,Z 660.616,A 0.000,B 0.000,C 90.000,E1 110.918} C_DIS
LIN {X 0.012,Y -391.131,Z 660.603,A 0.000,B 0.000,C 90.000,E1 108.598} C_DIS
LIN {X 0.183,Y -407.915,Z 660.591,A 0.000,B 0.000,C 90.000,E1 106.315} C_DIS
LIN {X 0.155,Y -426.336,Z 660.579,A 0.000,B 0.000,C 90.000,E1 104.120} C_DIS
LIN {X 0.215,Y -446.190,Z 660.567,A 0.000,B 0.000,C 90.000,E1 102.007} C_DIS
LIN {X 0.208,Y -466.657,Z 660.556,A 0.000,B 0.000,C 90.000,E1 100.074} C_DIS
LIN {X 0.180,Y -469.239,Z 660.555,A 0.000,B 0.000,C 90.000,E1 99.849} C_DIS
LIN {X 0.235,Y -471.490,Z 660.554,A 0.000,B 0.000,C 90.000,E1 99.613} C_DIS
LIN {X 0.117,Y -473.323,Z 660.552,A 0.000,B 0.000,C 90.000,E1 99.378} C_DIS
LIN {X -0.079,Y -474.704,Z 660.551,A 0.000,B 0.000,C 90.000,E1 99.151} C_DIS
LIN {X 0.114,Y -476.479,Z 660.548,A 0.000,B 0.000,C 90.000,E1 98.624} C_DIS
LIN {X -0.231,Y -477.167,Z 660.545,A 0.000,B 0.000,C 90.000,E1 98.163} C_DIS
LIN {X -0.091,Y -476.887,Z 660.542,A 0.000,B 0.000,C 90.000,E1 97.644} C_DIS
LIN {X 0.054,Y -475.596,Z 660.540,A 0.000,B 0.000,C 90.000,E1 97.125} C_DIS
LIN {X -0.081,Y -474.511,Z 660.538,A 0.000,B 0.000,C 90.000,E1 96.891} C_DIS
LIN {X 0.197,Y -473.056,Z 660.537,A 0.000,B 0.000,C 90.000,E1 96.606} C_DIS
LIN {X 0.135,Y -456.082,Z 660.523,A 0.000,B 0.000,C 90.000,E1 94.073} C_DIS
LIN {X 0.075,Y -443.951,Z 660.511,A 0.000,B 0.000,C 90.000,E1 92.007} C_DIS
LIN {X -0.161,Y -435.333,Z 660.502,A 0.000,B 0.000,C 90.000,E1 90.458} C_DIS
LIN {X 0.169,Y -427.948,Z 660.495,A 0.000,B 0.000,C 90.000,E1 89.083} C_DIS
LIN {X 0.192,Y -417.111,Z 660.485,A 0.000,B 0.000,C 90.000,E1 87.192} C_DIS
LIN {X 0.009,Y -406.179,Z 660.474,A 0.000,B 0.000,C 90.000,E1 85.298} C_DIS
LIN {X 0.170,Y -392.414,Z 660.460,A 0.000,B 0.000,C 90.000,E1 82.761} C_DIS
LIN {X 0.073,Y -379.129,Z 660.446,A 0.000,B 0.000,C 90.000,E1 80.208} C_DIS
LIN {X 0.071,Y -367.752,Z 660.433,A 0.000,B 0.000,C 90.000,E1 77.881} C_DIS
LIN {X -0.071,Y -354.070,Z 660.416,A 0.000,B 0.000,C 90.000,E1 74.936} C_DIS
LIN {X 0.082,Y -343.694,Z 660.403,A 0.000,B 0.000,C 90.000,E1 72.489} C_DIS
LIN {X 0.103,Y -329.062,Z 660.382,A 0.000,B 0.000,C 90.000,E1 68.773} C_DIS
LIN {X 0.032,Y -316.801,Z 660.363,A 0.000,B 0.000,C 90.000,E1 65.305} C_DIS
LIN {X 0.007,Y -304.981,Z 660.341,A 0.000,B 0.000,C 90.000,E1 61.435} C_DIS
LIN {X 0.143,Y -294.389,Z 660.319,A 0.000,B 0.000,C 90.000,E1 57.454} C_DIS
LIN {X -0.058,Y -287.800,Z 660.304,A 0.000,B 0.000,C 90.000,E1 54.815} C_DIS
LIN {X -0.081,Y -281.316,Z 660.289,A 0.000,B 0.000,C 90.000,E1 52.110} C_DIS
LIN {X 0.028,Y -276.246,Z 660.278,A 0.000,B 0.000,C 90.000,E1 50.033} C_DIS
LIN {X 0.034,Y -270.784,Z 660.266,A 0.000,B 0.000,C 90.000,E1 47.957} C_DIS
LIN {X -0.105,Y -264.917,Z 660.255,A 0.000,B 0.000,C 90.000,E1 45.891} C_DIS
LIN {X -0.160,Y -258.668,Z 660.243,A 0.000,B 0.000,C 90.000,E1 43.785} C_DIS
LIN {X 0.037,Y -252.166,Z 660.231,A 0.000,B 0.000,C 90.000,E1 41.595} C_DIS
LIN {X -0.017,Y -243.529,Z 660.215,A 0.000,B 0.000,C 90.000,E1 38.705} C_DIS
LIN {X 0.094,Y -235.434,Z 660.199,A 0.000,B 0.000,C 90.000,E1 35.724} C_DIS
LIN {X -0.030,Y -227.970,Z 660.182,A 0.000,B 0.000,C 90.000,E1 32.752} C_DIS
LIN {X 0.117,Y -221.200,Z 660.165,A 0.000,B 0.000,C 90.000,E1 29.667} C_DIS
LIN {X -0.038,Y -215.275,Z 660.148,A 0.000,B 0.000,C 90.000,E1 26.616} C_DIS
LIN {X 0.055,Y -210.195,Z 660.130,A 0.000,B 0.000,C 90.000,E1 23.462} C_DIS
LIN {X 0.054,Y -204.894,Z 660.108,A 0.000,B 0.000,C 90.000,E1 19.504} C_DIS
LIN {X -0.069,Y -200.701,Z 660.086,A 0.000,B 0.000,C 90.000,E1 15.536} C_DIS
LIN {X 0.034,Y -197.030,Z 660.059,A 0.000,B 0.000,C 90.000,E1 10.658} C_DIS
LIN {X 0.071,Y -194.401,Z 660.023,A 0.000,B 0.000,C 90.000,E1 4.131} C_DIS
LIN {X -0.014,Y -195.880,Z 659.961,A 0.000,B 0.000,C 90.000,E1 352.996} C_DIS
LIN {X -0.027,Y -198.911,Z 659.934,A 0.000,B 0.000,C 90.000,E1 348.117} C_DIS
LIN {X -0.118,Y -202.535,Z 659.911,A 0.000,B 0.000,C 90.000,E1 344.102} C_DIS
LIN {X 0.001,Y -207.165,Z 659.889,A 0.000,B 0.000,C 90.000,E1 340.061} C_DIS
LIN {X -0.023,Y -212.595,Z 659.867,A 0.000,B 0.000,C 90.000,E1 336.102} C_DIS
LIN {X 0.090,Y -218.813,Z 659.845,A 0.000,B 0.000,C 90.000,E1 332.153} C_DIS
LIN {X -0.068,Y -225.698,Z 659.824,A 0.000,B 0.000,C 90.000,E1 328.329} C_DIS
LIN {X 0.078,Y -233.116,Z 659.803,A 0.000,B 0.000,C 90.000,E1 324.482} C_DIS
LIN {X 0.118,Y -241.179,Z 659.782,A 0.000,B 0.000,C 90.000,E1 320.723} C_DIS
LIN {X -0.024,Y -250.034,Z 659.761,A 0.000,B 0.000,C 90.000,E1 317.067} C_DIS
LIN {X -0.092,Y -259.960,Z 659.741,A 0.000,B 0.000,C 90.000,E1 313.461} C_DIS
LIN {X -0.026,Y -269.972,Z 659.724,A 0.000,B 0.000,C 90.000,E1 310.253} C_DIS
LIN {X -0.079,Y -282.535,Z 659.704,A 0.000,B 0.000,C 90.000,E1 306.790} C_DIS
LIN {X 0.075,Y -293.507,Z 659.689,A 0.000,B 0.000,C 90.000,E1 304.040} C_DIS
LIN {X 0.082,Y -308.816,Z 659.671,A 0.000,B 0.000,C 90.000,E1 300.718} C_DIS
LIN {X -0.048,Y -325.497,Z 659.653,A 0.000,B 0.000,C 90.000,E1 297.513} C_DIS
LIN {X 0.096,Y -337.708,Z 659.641,A 0.000,B 0.000,C 90.000,E1 295.283} C_DIS
LIN {X 0.150,Y -356.022,Z 659.623,A 0.000,B 0.000,C 90.000,E1 292.206} C_DIS
LIN {X 0.106,Y -369.549,Z 659.612,A 0.000,B 0.000,C 90.000,E1 290.120} C_DIS
LIN {X 0.109,Y -382.396,Z 659.602,A 0.000,B 0.000,C 90.000,E1 288.362} C_DIS
LIN {X 0.148,Y -403.210,Z 659.588,A 0.000,B 0.000,C 90.000,E1 285.788} C_DIS
LIN {X 0.044,Y -414.804,Z 659.580,A 0.000,B 0.000,C 90.000,E1 284.411} C_DIS
LIN {X -0.108,Y -425.949,Z 659.573,A 0.000,B 0.000,C 90.000,E1 283.063} C_DIS
LIN {X 0.150,Y -434.416,Z 659.567,A 0.000,B 0.000,C 90.000,E1 281.951} C_DIS
LIN {X -0.131,Y -444.485,Z 659.559,A 0.000,B 0.000,C 90.000,E1 280.658} C_DIS
LIN {X -0.187,Y -456.488,Z 659.550,A 0.000,B 0.000,C 90.000,E1 279.095} C_DIS
LIN {X 0.095,Y -464.941,Z 659.545,A 0.000,B 0.000,C 90.000,E1 278.049} C_DIS
LIN {X 0.157,Y -468.937,Z 659.542,A 0.000,B 0.000,C 90.000,E1 277.530} C_DIS
LIN {X 0.088,Y -474.054,Z 659.538,A 0.000,B 0.000,C 90.000,E1 276.777} C_DIS
LIN {X 0.013,Y -478.330,Z 659.534,A 0.000,B 0.000,C 90.000,E1 276.030} C_DIS
LIN {X 0.020,Y -481.782,Z 659.529,A 0.000,B 0.000,C 90.000,E1 275.277} C_DIS
LIN {X 0.185,Y -483.601,Z 659.527,A 0.000,B 0.000,C 90.000,E1 274.759} C_DIS
LIN {X -0.165,Y -485.053,Z 659.524,A 0.000,B 0.000,C 90.000,E1 274.302} C_DIS
LIN {X 0.016,Y -486.083,Z 659.521,A 0.000,B 0.000,C 90.000,E1 273.784} C_DIS
LIN {X 0.175,Y -486.732,Z 659.518,A 0.000,B 0.000,C 90.000,E1 273.269} C_DIS
LIN {X -0.119,Y -487.068,Z 659.516,A 0.000,B 0.000,C 90.000,E1 272.808} C_DIS
LIN {X 0.053,Y -487.098,Z 659.513,A 0.000,B 0.000,C 90.000,E1 272.293} C_DIS
LIN {X 0.245,Y -486.870,Z 659.510,A 0.000,B 0.000,C 90.000,E1 271.776} C_DIS
LIN {X -0.066,Y -486.256,Z 659.507,A 0.000,B 0.000,C 90.000,E1 271.318} C_DIS
LIN {X 0.109,Y -485.242,Z 659.505,A 0.000,B 0.000,C 90.000,E1 270.802} C_DIS
LIN {X -0.203,Y -483.771,Z 659.502,A 0.000,B 0.000,C 90.000,E1 270.344} C_DIS
LIN {X -0.036,Y -481.768,Z 659.499,A 0.000,B 0.000,C 90.000,E1 269.828} C_DIS
LIN {X 0.121,Y -479.044,Z 659.496,A 0.000,B 0.000,C 90.000,E1 269.312} C_DIS
LIN {X -0.219,Y -475.519,Z 659.493,A 0.000,B 0.000,C 90.000,E1 268.854} C_DIS
LIN {X -0.101,Y -471.003,Z 659.491,A 0.000,B 0.000,C 90.000,E1 268.339} C_DIS
LIN {X 0.009,Y -465.279,Z 659.488,A 0.000,B 0.000,C 90.000,E1 267.822} C_DIS
LIN {X 0.065,Y -462.295,Z 659.487,A 0.000,B 0.000,C 90.000,E1 267.593} C_DIS
LIN {X 0.037,Y -455.735,Z 659.484,A 0.000,B 0.000,C 90.000,E1 267.192} C_DIS
LIN {X 0.122,Y -448.768,Z 659.483,A 0.000,B 0.000,C 90.000,E1 266.849} C_DIS
LIN {X -0.146,Y -441.259,Z 659.481,A 0.000,B 0.000,C 90.000,E1 266.617} C_DIS
LIN {X 0.058,Y -433.527,Z 659.480,A 0.000,B 0.000,C 90.000,E1 266.388} C_DIS
LIN {X -0.176,Y -424.448,Z 659.479,A 0.000,B 0.000,C 90.000,E1 266.274} C_DIS
LIN {X 0.155,Y -415.645,Z 659.479,A 0.000,B 0.000,C 90.000,E1 266.159} C_DIS
LIN {X 0.038,Y -180.928,Z 659.479,A 0.000,B 0.000,C 90.000,E1 266.159} C_DIS
LIN {X -0.077,Y -180.902,Z 659.474,A 0.000,B 0.000,C 90.000,E1 265.298} C_DIS
LIN {X 0.053,Y -180.232,Z 659.464,A 0.000,B 0.000,C 90.000,E1 263.571} C_DIS
LIN {X 0.068,Y -178.716,Z 659.441,A 0.000,B 0.000,C 90.000,E1 259.342} C_DIS
LIN {X -0.039,Y -175.764,Z 659.413,A 0.000,B 0.000,C 90.000,E1 254.283} C_DIS
LIN {X 0.011,Y -171.948,Z 659.384,A 0.000,B 0.000,C 90.000,E1 249.135} C_DIS
LIN {X -0.013,Y -171.336,Z 659.379,A 0.000,B 0.000,C 90.000,E1 248.284} C_DIS
LIN {X 0.039,Y -167.590,Z 659.355,A 0.000,B 0.000,C 90.000,E1 243.948} C_DIS
LIN {X -0.022,Y -166.228,Z 659.346,A 0.000,B 0.000,C 90.000,E1 242.231} C_DIS
LIN {X -0.033,Y -162.988,Z 659.326,A 0.000,B 0.000,C 90.000,E1 238.742} C_DIS
LIN {X 0.014,Y -160.906,Z 659.312,A 0.000,B 0.000,C 90.000,E1 236.087} C_DIS
LIN {X -0.008,Y -157.672,Z 659.292,A 0.000,B 0.000,C 90.000,E1 232.557} C_DIS
LIN {X -0.070,Y -155.709,Z 659.277,A 0.000,B 0.000,C 90.000,E1 229.908} C_DIS
LIN {X -0.015,Y -151.972,Z 659.252,A 0.000,B 0.000,C 90.000,E1 225.405} C_DIS
LIN {X 0.001,Y -150.215,Z 659.237,A 0.000,B 0.000,C 90.000,E1 222.690} C_DIS
LIN {X -0.075,Y -146.979,Z 659.212,A 0.000,B 0.000,C 90.000,E1 218.177} C_DIS
LIN {X 0.034,Y -145.566,Z 659.197,A 0.000,B 0.000,C 90.000,E1 215.391} C_DIS
LIN {X 0.034,Y -142.957,Z 659.171,A 0.000,B 0.000,C 90.000,E1 210.797} C_DIS
LIN {X -0.036,Y -141.583,Z 659.151,A 0.000,B 0.000,C 90.000,E1 207.129} C_DIS
LIN {X 0.011,Y -139.417,Z 659.115,A 0.000,B 0.000,C 90.000,E1 200.610} C_DIS
LIN {X 0.063,Y -139.142,Z 659.104,A 0.000,B 0.000,C 90.000,E1 198.725} C_DIS
LIN {X -0.046,Y -138.348,Z 659.057,A 0.000,B 0.000,C 90.000,E1 190.366} C_DIS
LIN {X -0.061,Y -139.490,Z 659.006,A 0.000,B 0.000,C 90.000,E1 181.031} C_DIS
LIN {X 0.020,Y -141.100,Z 658.975,A 0.000,B 0.000,C 90.000,E1 175.412} C_DIS
LIN {X -0.027,Y -142.479,Z 658.959,A 0.000,B 0.000,C 90.000,E1 172.648} C_DIS
LIN {X 0.062,Y -144.727,Z 658.933,A 0.000,B 0.000,C 90.000,E1 167.993} C_DIS
LIN {X 0.013,Y -147.331,Z 658.913,A 0.000,B 0.000,C 90.000,E1 164.338} C_DIS
LIN {X 0.078,Y -150.653,Z 658.888,A 0.000,B 0.000,C 90.000,E1 159.752} C_DIS
LIN {X -0.040,Y -154.131,Z 658.868,A 0.000,B 0.000,C 90.000,E1 156.177} C_DIS
LIN {X 0.022,Y -157.559,Z 658.848,A 0.000,B 0.000,C 90.000,E1 152.564} C_DIS
LIN {X 0.047,Y -161.801,Z 658.828,A 0.000,B 0.000,C 90.000,E1 148.997} C_DIS
LIN {X 0.067,Y -165.993,Z 658.808,A 0.000,B 0.000,C 90.000,E1 145.468} C_DIS
LIN {X 0.060,Y -170.990,Z 658.789,A 0.000,B 0.000,C 90.000,E1 141.984} C_DIS
LIN {X -0.025,Y -175.859,Z 658.770,A 0.000,B 0.000,C 90.000,E1 138.566} C_DIS
LIN {X -0.030,Y -181.465,Z 658.751,A 0.000,B 0.000,C 90.000,E1 135.162} C_DIS
LIN {X 0.106,Y -186.975,Z 658.732,A 0.000,B 0.000,C 90.000,E1 131.757} C_DIS
LIN {X 0.120,Y -191.057,Z 658.720,A 0.000,B 0.000,C 90.000,E1 129.564} C_DIS
LIN {X 0.129,Y -289.312,Z 658.720,A 0.000,B 0.000,C 90.000,E1 129.564} C_DIS
LIN {X 0.024,Y -290.390,Z 658.720,A 0.000,B 0.000,C 90.000,E1 129.564} C_DIS
LIN {X 0.095,Y -295.667,Z 658.718,A 0.000,B 0.000,C 90.000,E1 129.277} C_DIS
LIN {X -0.075,Y -298.830,Z 658.717,A 0.000,B 0.000,C 90.000,E1 128.991} C_DIS
LIN {X 0.116,Y -302.449,Z 658.713,A 0.000,B 0.000,C 90.000,E1 128.382} C_DIS
LIN {X -0.123,Y -303.916,Z 658.711,A 0.000,B 0.000,C 90.000,E1 128.096} C_DIS
LIN {X 0.064,Y -305.070,Z 658.710,A 0.000,B 0.000,C 90.000,E1 127.729} C_DIS
LIN {X 0.176,Y -315.629,Z 658.690,A 0.000,B 0.000,C 90.000,E1 124.119} C_DIS
LIN {X 0.056,Y -325.595,Z 658.674,A 0.000,B 0.000,C 90.000,E1 121.258} C_DIS
LIN {X 0.004,Y -336.882,Z 658.658,A 0.000,B 0.000,C 90.000,E1 118.437} C_DIS
LIN {X -0.042,Y -349.593,Z 658.643,A 0.000,B 0.000,C 90.000,E1 115.668} C_DIS
LIN {X -0.094,Y -362.178,Z 658.629,A 0.000,B 0.000,C 90.000,E1 113.259} C_DIS
LIN {X 0.082,Y -376.067,Z 658.616,A 0.000,B 0.000,C 90.000,E1 110.865} C_DIS
LIN {X 0.135,Y -391.360,Z 658.603,A 0.000,B 0.000,C 90.000,E1 108.544} C_DIS
LIN {X -0.069,Y -408.169,Z 658.591,A 0.000,B 0.000,C 90.000,E1 106.315} C_DIS
LIN {X -0.103,Y -426.617,Z 658.578,A 0.000,B 0.000,C 90.000,E1 104.120} C_DIS
LIN {X -0.036,Y -446.485,Z 658.567,A 0.000,B 0.000,C 90.000,E1 102.007} C_DIS
LIN {X -0.035,Y -466.961,Z 658.556,A 0.000,B 0.000,C 90.000,E1 100.074} C_DIS
LIN {X -0.060,Y -469.541,Z 658.555,A 0.000,B 0.000,C 90.000,E1 99.849} C_DIS
LIN {X -0.005,Y -471.732,Z 658.553,A 0.000,B 0.000,C 90.000,E1 99.613} C_DIS
LIN {X -0.153,Y -473.546,Z 658.552,A 0.000,B 0.000,C 90.000,E1 99.378} C_DIS
LIN {X 0.091,Y -474.907,Z 658.551,A 0.000,B 0.000,C 90.000,E1 99.095} C_DIS
LIN {X -0.186,Y -476.618,Z 658.548,A 0.000,B 0.000,C 90.000,E1 98.624} C_DIS
LIN {X -0.057,Y -477.254,Z 658.545,A 0.000,B 0.000,C 90.000,E1 98.106} C_DIS
LIN {X 0.084,Y -476.922,Z 658.542,A 0.000,B 0.000,C 90.000,E1 97.587} C_DIS
LIN {X -0.242,Y -475.574,Z 658.539,A 0.000,B 0.000,C 90.000,E1 97.125} C_DIS
LIN {X 0.095,Y -474.453,Z 658.538,A 0.000,B 0.000,C 90.000,E1 96.834} C_DIS
LIN {X -0.096,Y -472.954,Z 658.537,A 0.000,B 0.000,C 90.000,E1 96.606} C_DIS
LIN {X -0.151,Y -455.957,Z 658.523,A 0.000,B 0.000,C 90.000,E1 94.073} C_DIS
LIN {X -0.206,Y -443.835,Z 658.511,A 0.000,B 0.000,C 90.000,E1 92.007} C_DIS
LIN {X -0.004,Y -435.226,Z 658.502,A 0.000,B 0.000,C 90.000,E1 90.401} C_DIS
LIN {X -0.105,Y -427.841,Z 658.495,A 0.000,B 0.000,C 90.000,E1 89.083} C_DIS
LIN {X -0.078,Y -417.001,Z 658.484,A 0.000,B 0.000,C 90.000,E1 87.192} C_DIS
LIN {X 0.148,Y -406.061,Z 658.474,A 0.000,B 0.000,C 90.000,E1 85.241} C_DIS
LIN {X -0.089,Y -392.320,Z 658.460,A 0.000,B 0.000,C 90.000,E1 82.761} C_DIS
LIN {X 0.194,Y -379.060,Z 658.445,A 0.000,B 0.000,C 90.000,E1 80.151} C_DIS
LIN {X -0.175,Y -367.697,Z 658.432,A 0.000,B 0.000,C 90.000,E1 77.881} C_DIS
LIN {X 0.124,Y -354.045,Z 658.416,A 0.000,B 0.000,C 90.000,E1 74.866} C_DIS
LIN {X -0.151,Y -343.695,Z 658.403,A 0.000,B 0.000,C 90.000,E1 72.489} C_DIS
LIN {X -0.118,Y -329.106,Z 658.382,A 0.000,B 0.000,C 90.000,E1 68.773} C_DIS
LIN {X -0.046,Y -316.881,Z 658.363,A 0.000,B 0.000,C 90.000,E1 65.281} C_DIS
LIN {X 0.074,Y -305.080,Z 658.341,A 0.000,B 0.000,C 90.000,E1 61.385} C_DIS
LIN {X -0.045,Y -294.498,Z 658.319,A 0.000,B 0.000,C 90.000,E1 57.454} C_DIS
LIN {X -0.005,Y -287.892,Z 658.304,A 0.000,B 0.000,C 90.000,E1 54.769} C_DIS
LIN {X -0.035,Y -281.440,Z 658.289,A 0.000,B 0.000,C 90.000,E1 52.065} C_DIS
LIN {X 0.058,Y -278.122,Z 658.282,A 0.000,B 0.000,C 90.000,E1 50.678} C_DIS
LIN {X 0.067,Y -272.764,Z 658.270,A 0.000,B 0.000,C 90.000,E1 48.609} C_DIS
LIN {X -0.018,Y -267.041,Z 658.259,A 0.000,B 0.000,C 90.000,E1 46.539} C_DIS
LIN {X -0.037,Y -260.883,Z 658.247,A 0.000,B 0.000,C 90.000,E1 44.433} C_DIS
LIN {X 0.015,Y -254.437,Z 658.235,A 0.000,B 0.000,C 90.000,E1 42.285} C_DIS
LIN {X -0.018,Y -245.721,Z 658.219,A 0.000,B 0.000,C 90.000,E1 39.402} C_DIS
LIN {X 0.001,Y -237.460,Z 658.203,A 0.000,B 0.000,C 90.000,E1 36.457} C_DIS
LIN {X 0.064,Y -229.862,Z 658.186,A 0.000,B 0.000,C 90.000,E1 33.452} C_DIS
LIN {X -0.121,Y -222.896,Z 658.169,A 0.000,B 0.000,C 90.000,E1 30.463} C_DIS
LIN {X 0.066,Y -216.775,Z 658.152,A 0.000,B 0.000,C 90.000,E1 27.334} C_DIS
LIN {X 0.094,Y -211.495,Z 658.135,A 0.000,B 0.000,C 90.000,E1 24.207} C_DIS
LIN {X -0.060,Y -205.962,Z 658.113,A 0.000,B 0.000,C 90.000,E1 20.301} C_DIS
LIN {X -0.084,Y -201.553,Z 658.091,A 0.000,B 0.000,C 90.000,E1 16.315} C_DIS
LIN {X -0.093,Y -197.637,Z 658.064,A 0.000,B 0.000,C 90.000,E1 11.478} C_DIS
LIN {X 0.064,Y -194.917,Z 658.032,A 0.000,B 0.000,C 90.000,E1 5.739} C_DIS
LIN {X -0.010,Y -195.955,Z 657.961,A 0.000,B 0.000,C 90.000,E1 352.996} C_DIS
LIN {X -0.020,Y -198.991,Z 657.934,A 0.000,B 0.000,C 90.000,E1 348.117} C_DIS
LIN {X -0.109,Y -202.594,Z 657.911,A 0.000,B 0.000,C 90.000,E1 344.102} C_DIS
LIN {X 0.012,Y -207.224,Z 657.889,A 0.000,B 0.000,C 90.000,E1 340.061} C_DIS
LIN {X -0.009,Y -212.651,Z 657.867,A 0.000,B 0.000,C 90.000,E1 336.102} C_DIS
LIN {X 0.107,Y -218.857,Z 657.845,A 0.000,B 0.000,C 90.000,E1 332.153} C_DIS
LIN {X -0.050,Y -225.745,Z 657.824,A 0.000,B 0.000,C 90.000,E1 328.329} C_DIS
LIN {X 0.099,Y -233.138,Z 657.803,A 0.000,B 0.000,C 90.000,E1 324.482} C_DIS
LIN {X 0.140,Y -241.180,Z 657.782,A 0.000,B 0.000,C 90.000,E1 320.723} C_DIS
LIN {X -0.001,Y -250.025,Z 657.761,A 0.000,B 0.000,C 90.000,E1 317.067} C_DIS
LIN {X -0.068,Y -259.935,Z 657.741,A 0.000,B 0.000,C 90.000,E1 313.461} C_DIS
LIN {X -0.075,Y -268.741,Z 657.726,A 0.000,B 0.000,C 90.000,E1 310.620} C_DIS
LIN {X -0.170,Y -281.155,Z 657.706,A 0.000,B 0.000,C 90.000,E1 307.156} C_DIS
LIN {X -0.067,Y -293.435,Z 657.689,A 0.000,B 0.000,C 90.000,E1 304.072} C_DIS
LIN {X 0.102,Y -308.734,Z 657.671,A 0.000,B 0.000,C 90.000,E1 300.718} C_DIS
LIN {X -0.029,Y -325.430,Z 657.653,A 0.000,B 0.000,C 90.000,E1 297.513} C_DIS
LIN {X 0.099,Y -339.387,Z 657.639,A 0.000,B 0.000,C 90.000,E1 294.975} C_DIS
LIN {X 0.212,Y -357.817,Z 657.622,A 0.000,B 0.000,C 90.000,E1 291.897} C_DIS
LIN {X 0.121,Y -369.459,Z 657.612,A 0.000,B 0.000,C 90.000,E1 290.120} C_DIS
LIN {X 0.123,Y -382.294,Z 657.602,A 0.000,B 0.000,C 90.000,E1 288.362} C_DIS
LIN {X 0.161,Y -403.110,Z 657.588,A 0.000,B 0.000,C 90.000,E1 285.788} C_DIS
LIN {X 0.055,Y -414.690,Z 657.580,A 0.000,B 0.000,C 90.000,E1 284.411} C_DIS
LIN {X -0.098,Y -425.833,Z 657.573,A 0.000,B 0.000,C 90.000,E1 283.063} C_DIS
LIN {X 0.159,Y -434.310,Z 657.567,A 0.000,B 0.000,C 90.000,E1 281.951} C_DIS
LIN {X -0.124,Y -444.410,Z 657.559,A 0.000,B 0.000,C 90.000,E1 280.658} C_DIS
LIN {X -0.158,Y -456.403,Z 657.550,A 0.000,B 0.000,C 90.000,E1 279.095} C_DIS
LIN {X 0.138,Y -464.912,Z 657.545,A 0.000,B 0.000,C 90.000,E1 278.049} C_DIS
LIN {X 0.199,Y -468.842,Z 657.542,A 0.000,B 0.000,C 90.000,E1 277.530} C_DIS
LIN {X -0.182,Y -472.393,Z 657.539,A 0.000,B 0.000,C 90.000,E1 277.068} C_DIS
LIN {X -0.226,Y -476.912,Z 657.535,A 0.000,B 0.000,C 90.000,E1 276.315} C_DIS
LIN {X 0.200,Y -480.697,Z 657.531,A 0.000,B 0.000,C 90.000,E1 275.511} C_DIS
LIN {X 0.226,Y -483.562,Z 657.527,A 0.000,B 0.000,C 90.000,E1 274.759} C_DIS
LIN {X -0.124,Y -484.997,Z 657.524,A 0.000,B 0.000,C 90.000,E1 274.302} C_DIS
LIN {X 0.057,Y -486.018,Z 657.521,A 0.000,B 0.000,C 90.000,E1 273.784} C_DIS
LIN {X 0.216,Y -486.670,Z 657.518,A 0.000,B 0.000,C 90.000,E1 273.269} C_DIS
LIN {X -0.079,Y -487.025,Z 657.516,A 0.000,B 0.000,C 90.000,E1 272.808} C_DIS
LIN {X 0.093,Y -487.069,Z 657.513,A 0.000,B 0.000,C 90.000,E1 272.293} C_DIS
LIN {X -0.201,Y -486.834,Z 657.510,A 0.000,B 0.000,C 90.000,E1 271.833} C_DIS
LIN {X -0.027,Y -486.238,Z 657.507,A 0.000,B 0.000,C 90.000,E1 271.318} C_DIS
LIN {X 0.149,Y -485.258,Z 657.505,A 0.000,B 0.000,C 90.000,E1 270.802} C_DIS
LIN {X -0.164,Y -483.778,Z 657.502,A 0.000,B 0.000,C 90.000,E1 270.344} C_DIS
LIN {X 0.003,Y -481.773,Z 657.499,A 0.000,B 0.000,C 90.000,E1 269.828} C_DIS
LIN {X 0.160,Y -479.073,Z 657.496,A 0.000,B 0.000,C 90.000,E1 269.312} C_DIS
LIN {X -0.181,Y -475.566,Z 657.494,A 0.000,B 0.000,C 90.000,E1 268.854} C_DIS
LIN {X 0.116,Y -473.471,Z 657.492,A 0.000,B 0.000,C 90.000,E1 268.568} C_DIS
LIN {X 0.234,Y -468.389,Z 657.489,A 0.000,B 0.000,C 90.000,E1 268.051} C_DIS
LIN {X 0.047,Y -465.387,Z 657.488,A 0.000,B 0.000,C 90.000,E1 267.822} C_DIS
LIN {X 0.107,Y -462.419,Z 657.487,A 0.000,B 0.000,C 90.000,E1 267.593} C_DIS
LIN {X 0.165,Y -459.051,Z 657.485,A 0.000,B 0.000,C 90.000,E1 267.364} C_DIS
LIN {X -0.065,Y -452.154,Z 657.483,A 0.000,B 0.000,C 90.000,E1 267.020} C_DIS
LIN {X -0.168,Y -444.782,Z 657.482,A 0.000,B 0.000,C 90.000,E1 266.731} C_DIS
LIN {X 0.216,Y -436.860,Z 657.480,A 0.000,B 0.000,C 90.000,E1 266.445} C_DIS
LIN {X -0.197,Y -428.812,Z 657.479,A 0.000,B 0.000,C 90.000,E1 266.331} C_DIS
LIN {X 0.179,Y -417.667,Z 657.479,A 0.000,B 0.000,C 90.000,E1 266.159} C_DIS
LIN {X 0.112,Y -414.413,Z 657.479,A 0.000,B 0.000,C 90.000,E1 266.159} C_DIS
LIN {X 0.020,Y -180.928,Z 657.479,A 0.000,B 0.000,C 90.000,E1 266.159} C_DIS
LIN {X -0.095,Y -180.902,Z 657.474,A 0.000,B 0.000,C 90.000,E1 265.298} C_DIS
LIN {X 0.034,Y -180.229,Z 657.464,A 0.000,B 0.000,C 90.000,E1 263.571} C_DIS
LIN {X -0.013,Y -179.042,Z 657.446,A 0.000,B 0.000,C 90.000,E1 260.208} C_DIS
LIN {X 0.050,Y -178.712,Z 657.441,A 0.000,B 0.000,C 90.000,E1 259.342} C_DIS
LIN {X -0.057,Y -175.761,Z 657.413,A 0.000,B 0.000,C 90.000,E1 254.283} C_DIS
LIN {X -0.007,Y -171.945,Z 657.384,A 0.000,B 0.000,C 90.000,E1 249.135} C_DIS
LIN {X -0.031,Y -171.330,Z 657.379,A 0.000,B 0.000,C 90.000,E1 248.284} C_DIS
LIN {X 0.021,Y -167.585,Z 657.355,A 0.000,B 0.000,C 90.000,E1 243.948} C_DIS
LIN {X -0.039,Y -166.222,Z 657.346,A 0.000,B 0.000,C 90.000,E1 242.231} C_DIS
LIN {X -0.050,Y -162.984,Z 657.326,A 0.000,B 0.000,C 90.000,E1 238.742} C_DIS
LIN {X -0.004,Y -160.900,Z 657.312,A 0.000,B 0.000,C 90.000,E1 236.087} C_DIS
LIN {X -0.025,Y -157.666,Z 657.292,A 0.000,B 0.000,C 90.000,E1 232.557} C_DIS
LIN {X -0.087,Y -155.704,Z 657.277,A 0.000,B 0.000,C 90.000,E1 229.908} C_DIS
LIN {X -0.032,Y -151.967,Z 657.252,A 0.000,B 0.000,C 90.000,E1 225.405} C_DIS
LIN {X -0.015,Y -150.209,Z 657.237,A 0.000,B 0.000,C 90.000,E1 222.690} C_DIS
LIN {X -0.091,Y -146.975,Z 657.212,A 0.000,B 0.000,C 90.000,E1 218.177} C_DIS
LIN {X 0.019,Y -145.562,Z 657.197,A 0.000,B 0.000,C 90.000,E1 215.391} C_DIS
LIN {X 0.017,Y -142.954,Z 657.171,A 0.000,B 0.000,C 90.000,E1 210.797} C_DIS
LIN {X -0.052,Y -141.579,Z 657.151,A 0.000,B 0.000,C 90.000,E1 207.129} C_DIS
LIN {X -0.005,Y -139.416,Z 657.115,A 0.000,B 0.000,C 90.000,E1 200.610} C_DIS
LIN {X 0.048,Y -139.140,Z 657.104,A 0.000,B 0.000,C 90.000,E1 198.725} C_DIS
LIN {X -0.062,Y -138.348,Z 657.057,A 0.000,B 0.000,C 90.000,E1 190.366} C_DIS
LIN {X 0.063,Y -139.492,Z 657.006,A 0.000,B 0.000,C 90.000,E1 180.974} C_DIS
LIN {X 0.004,Y -141.103,Z 656.975,A 0.000,B 0.000,C 90.000,E1 175.412} C_DIS
LIN {X -0.043,Y -142.482,Z 656.959,A 0.000,B 0.000,C 90.000,E1 172.648} C_DIS
LIN {X 0.046,Y -144.731,Z 656.933,A 0.000,B 0.000,C 90.000,E1 167.993} C_DIS
LIN {X -0.004,Y -147.336,Z 656.913,A 0.000,B 0.000,C 90.000,E1 164.338} C_DIS
LIN {X 0.061,Y -150.659,Z 656.888,A 0.000,B 0.000,C 90.000,E1 159.752} C_DIS
LIN {X -0.057,Y -154.137,Z 656.868,A 0.000,B 0.000,C 90.000,E1 156.177} C_DIS
LIN {X 0.006,Y -157.565,Z 656.848,A 0.000,B 0.000,C 90.000,E1 152.564} C_DIS
LIN {X 0.029,Y -161.809,Z 656.828,A 0.000,B 0.000,C 90.000,E1 148.997} C_DIS
LIN {X 0.049,Y -166.000,Z 656.808,A 0.000,B 0.000,C 90.000,E1 145.468} C_DIS
LIN {X 0.042,Y -170.999,Z 656.789,A 0.000,B 0.000,C 90.000,E1 141.984} C_DIS
LIN {X -0.043,Y -175.869,Z 656.770,A 0.000,B 0.000,C 90.000,E1 138.566} C_DIS
LIN {X -0.049,Y -181.474,Z 656.751,A 0.000,B 0.000,C 90.000,E1 135.162} C_DIS
LIN {X 0.087,Y -186.986,Z 656.732,A 0.000,B 0.000,C 90.000,E1 131.757} C_DIS
LIN {X 0.014,Y -191.049,Z 656.720,A 0.000,B 0.000,C 90.000,E1 129.600} C_DIS
LIN {X 0.153,Y -289.173,Z 656.720,A 0.000,B 0.000,C 90.000,E1 129.564} C_DIS
LIN {X -0.004,Y -290.701,Z 656.720,A 0.000,B 0.000,C 90.000,E1 129.564} C_DIS
LIN {X 0.066,Y -295.752,Z 656.718,A 0.000,B 0.000,C 90.000,E1 129.277} C_DIS
LIN {X 0.011,Y -298.984,Z 656.716,A 0.000,B 0.000,C 90.000,E1 128.955} C_DIS
LIN {X -0.034,Y -302.578,Z 656.713,A 0.000,B 0.000,C 90.000,E1 128.382} C_DIS
LIN {X 0.153,Y -304.010,Z 656.711,A 0.000,B 0.000,C 90.000,E1 128.016} C_DIS
LIN {X -0.087,Y -305.137,Z 656.710,A 0.000,B 0.000,C 90.000,E1 127.729} C_DIS
LIN {X 0.024,Y -315.697,Z 656.690,A 0.000,B 0.000,C 90.000,E1 124.119} C_DIS
LIN {X -0.100,Y -325.676,Z 656.674,A 0.000,B 0.000,C 90.000,E1 121.258} C_DIS
LIN {X 0.005,Y -336.975,Z 656.658,A 0.000,B 0.000,C 90.000,E1 118.409} C_DIS
LIN {X -0.052,Y -349.701,Z 656.642,A 0.000,B 0.000,C 90.000,E1 115.643} C_DIS
LIN {X 0.074,Y -362.298,Z 656.629,A 0.000,B 0.000,C 90.000,E1 113.206} C_DIS
LIN {X 0.048,Y -376.202,Z 656.616,A 0.000,B 0.000,C 90.000,E1 110.844} C_DIS
LIN {X -0.037,Y -391.511,Z 656.603,A 0.000,B 0.000,C 90.000,E1 108.544} C_DIS
LIN {X 0.148,Y -408.337,Z 656.590,A 0.000,B 0.000,C 90.000,E1 106.260} C_DIS
LIN {X 0.132,Y -426.803,Z 656.578,A 0.000,B 0.000,C 90.000,E1 104.064} C_DIS
LIN {X -0.212,Y -446.681,Z 656.567,A 0.000,B 0.000,C 90.000,E1 102.007} C_DIS
LIN {X 0.256,Y -467.163,Z 656.556,A 0.000,B 0.000,C 90.000,E1 100.018} C_DIS
LIN {X -0.229,Y -469.741,Z 656.555,A 0.000,B 0.000,C 90.000,E1 99.849} C_DIS
LIN {X -0.172,Y -471.900,Z 656.553,A 0.000,B 0.000,C 90.000,E1 99.613} C_DIS
LIN {X 0.147,Y -473.690,Z 656.552,A 0.000,B 0.000,C 90.000,E1 99.321} C_DIS
LIN {X -0.076,Y -475.036,Z 656.550,A 0.000,B 0.000,C 90.000,E1 99.095} C_DIS
LIN {X 0.118,Y -476.723,Z 656.548,A 0.000,B 0.000,C 90.000,E1 98.568} C_DIS
LIN {X -0.224,Y -477.340,Z 656.545,A 0.000,B 0.000,C 90.000,E1 98.106} C_DIS
LIN {X -0.082,Y -476.989,Z 656.542,A 0.000,B 0.000,C 90.000,E1 97.587} C_DIS
LIN {X 0.066,Y -475.620,Z 656.539,A 0.000,B 0.000,C 90.000,E1 97.068} C_DIS
LIN {X -0.070,Y -474.484,Z 656.538,A 0.000,B 0.000,C 90.000,E1 96.834} C_DIS
LIN {X 0.066,Y -471.202,Z 656.535,A 0.000,B 0.000,C 90.000,E1 96.315} C_DIS
LIN {X -0.052,Y -454.335,Z 656.521,A 0.000,B 0.000,C 90.000,E1 93.784} C_DIS
LIN {X 0.027,Y -440.959,Z 656.508,A 0.000,B 0.000,C 90.000,E1 91.432} C_DIS
LIN {X 0.165,Y -432.280,Z 656.499,A 0.000,B 0.000,C 90.000,E1 89.828} C_DIS
LIN {X 0.016,Y -424.762,Z 656.492,A 0.000,B 0.000,C 90.000,E1 88.511} C_DIS
LIN {X -0.004,Y -413.881,Z 656.481,A 0.000,B 0.000,C 90.000,E1 86.617} C_DIS
LIN {X -0.027,Y -398.375,Z 656.466,A 0.000,B 0.000,C 90.000,E1 83.856} C_DIS
LIN {X -0.073,Y -384.916,Z 656.452,A 0.000,B 0.000,C 90.000,E1 81.319} C_DIS
LIN {X 0.067,Y -370.555,Z 656.436,A 0.000,B 0.000,C 90.000,E1 78.409} C_DIS
LIN {X 0.052,Y -358.104,Z 656.421,A 0.000,B 0.000,C 90.000,E1 75.755} C_DIS
LIN {X -0.201,Y -346.318,Z 656.406,A 0.000,B 0.000,C 90.000,E1 73.087} C_DIS
LIN {X 0.126,Y -331.552,Z 656.385,A 0.000,B 0.000,C 90.000,E1 69.337} C_DIS
LIN {X -0.165,Y -319.140,Z 656.366,A 0.000,B 0.000,C 90.000,E1 65.921} C_DIS
LIN {X 0.040,Y -307.112,Z 656.345,A 0.000,B 0.000,C 90.000,E1 62.025} C_DIS
LIN {X 0.102,Y -296.336,Z 656.323,A 0.000,B 0.000,C 90.000,E1 58.074} C_DIS
LIN {X -0.055,Y -289.691,Z 656.308,A 0.000,B 0.000,C 90.000,E1 55.435} C_DIS
LIN {X 0.028,Y -283.223,Z 656.293,A 0.000,B 0.000,C 90.000,E1 52.718} C_DIS
LIN {X -0.011,Y -278.288,Z 656.282,A 0.000,B 0.000,C 90.000,E1 50.678} C_DIS
LIN {X 0.003,Y -272.944,Z 656.270,A 0.000,B 0.000,C 90.000,E1 48.609} C_DIS
LIN {X -0.078,Y -267.215,Z 656.258,A 0.000,B 0.000,C 90.000,E1 46.539} C_DIS
LIN {X -0.092,Y -261.049,Z 656.247,A 0.000,B 0.000,C 90.000,E1 44.433} C_DIS
LIN {X -0.036,Y -254.583,Z 656.235,A 0.000,B 0.000,C 90.000,E1 42.285} C_DIS
LIN {X -0.063,Y -245.845,Z 656.219,A 0.000,B 0.000,C 90.000,E1 39.402} C_DIS
LIN {X -0.079,Y -235.614,Z 656.198,A 0.000,B 0.000,C 90.000,E1 35.724} C_DIS
LIN {X -0.001,Y -228.201,Z 656.182,A 0.000,B 0.000,C 90.000,E1 32.704} C_DIS
LIN {X -0.036,Y -221.427,Z 656.165,A 0.000,B 0.000,C 90.000,E1 29.667} C_DIS
LIN {X 0.012,Y -215.527,Z 656.148,A 0.000,B 0.000,C 90.000,E1 26.565} C_DIS
LIN {X -0.079,Y -210.424,Z 656.130,A 0.000,B 0.000,C 90.000,E1 23.462} C_DIS
LIN {X -0.069,Y -205.097,Z 656.108,A 0.000,B 0.000,C 90.000,E1 19.504} C_DIS
LIN {X 0.009,Y -200.903,Z 656.086,A 0.000,B 0.000,C 90.000,E1 15.481} C_DIS
LIN {X -0.071,Y -197.220,Z 656.059,A 0.000,B 0.000,C 90.000,E1 10.658} C_DIS
LIN {X -0.024,Y -194.585,Z 656.023,A 0.000,B 0.000,C 90.000,E1 4.131} C_DIS
LIN {X -0.006,Y -196.029,Z 655.961,A 0.000,B 0.000,C 90.000,E1 352.996} C_DIS
LIN {X -0.013,Y -199.069,Z 655.934,A 0.000,B 0.000,C 90.000,E1 348.117} C_DIS
LIN {X -0.099,Y -202.656,Z 655.911,A 0.000,B 0.000,C 90.000,E1 344.102} C_DIS
LIN {X 0.024,Y -207.280,Z 655.889,A 0.000,B 0.000,C 90.000,E1 340.061} C_DIS
LIN {X 0.005,Y -212.708,Z 655.867,A 0.000,B 0.000,C 90.000,E1 336.102} C_DIS
LIN {X 0.123,Y -218.898,Z 655.845,A 0.000,B 0.000,C 90.000,E1 332.153} C_DIS
LIN {X -0.032,Y -225.789,Z 655.824,A 0.000,B 0.000,C 90.000,E1 328.329} C_DIS
LIN {X 0.118,Y -233.169,Z 655.803,A 0.000,B 0.000,C 90.000,E1 324.482} C_DIS
LIN {X 0.008,Y -241.189,Z 655.782,A 0.000,B 0.000,C 90.000,E1 320.759} C_DIS
LIN {X 0.022,Y -250.026,Z 655.762,A 0.000,B 0.000,C 90.000,E1 317.067} C_DIS
LIN {X -0.045,Y -259.899,Z 655.741,A 0.000,B 0.000,C 90.000,E1 313.461} C_DIS
LIN {X -0.052,Y -268.677,Z 655.726,A 0.000,B 0.000,C 90.000,E1 310.620} C_DIS
LIN {X -0.148,Y -281.087,Z 655.706,A 0.000,B 0.000,C 90.000,E1 307.156} C_DIS
LIN {X -0.046,Y -293.362,Z 655.689,A 0.000,B 0.000,C 90.000,E1 304.072} C_DIS
LIN {X -0.035,Y -308.650,Z 655.671,A 0.000,B 0.000,C 90.000,E1 300.747} C_DIS
LIN {X -0.010,Y -325.355,Z 655.653,A 0.000,B 0.000,C 90.000,E1 297.513} C_DIS
LIN {X -0.190,Y -339.306,Z 655.639,A 0.000,B 0.000,C 90.000,E1 295.027} C_DIS
LIN {X 0.183,Y -355.829,Z 655.624,A 0.000,B 0.000,C 90.000,E1 292.206} C_DIS
LIN {X 0.137,Y -369.370,Z 655.612,A 0.000,B 0.000,C 90.000,E1 290.120} C_DIS
LIN {X 0.137,Y -382.187,Z 655.602,A 0.000,B 0.000,C 90.000,E1 288.362} C_DIS
LIN {X 0.106,Y -400.661,Z 655.589,A 0.000,B 0.000,C 90.000,E1 286.079} C_DIS
LIN {X -0.151,Y -412.333,Z 655.582,A 0.000,B 0.000,C 90.000,E1 284.717} C_DIS
LIN {X 0.178,Y -423.527,Z 655.574,A 0.000,B 0.000,C 90.000,E1 283.300} C_DIS
LIN {X 0.167,Y -434.218,Z 655.567,A 0.000,B 0.000,C 90.000,E1 281.951} C_DIS
LIN {X -0.117,Y -444.365,Z 655.559,A 0.000,B 0.000,C 90.000,E1 280.658} C_DIS
LIN {X 0.090,Y -454.256,Z 655.552,A 0.000,B 0.000,C 90.000,E1 279.321} C_DIS
LIN {X -0.201,Y -464.773,Z 655.545,A 0.000,B 0.000,C 90.000,E1 278.106} C_DIS
LIN {X 0.156,Y -470.530,Z 655.541,A 0.000,B 0.000,C 90.000,E1 277.296} C_DIS
LIN {X 0.048,Y -475.344,Z 655.536,A 0.000,B 0.000,C 90.000,E1 276.549} C_DIS
LIN {X 0.031,Y -479.380,Z 655.532,A 0.000,B 0.000,C 90.000,E1 275.796} C_DIS
LIN {X 0.183,Y -481.600,Z 655.529,A 0.000,B 0.000,C 90.000,E1 275.277} C_DIS
LIN {X -0.174,Y -483.447,Z 655.527,A 0.000,B 0.000,C 90.000,E1 274.821} C_DIS
LIN {X -0.003,Y -484.878,Z 655.524,A 0.000,B 0.000,C 90.000,E1 274.302} C_DIS
LIN {X 0.179,Y -485.960,Z 655.521,A 0.000,B 0.000,C 90.000,E1 273.784} C_DIS
LIN {X -0.150,Y -486.634,Z 655.518,A 0.000,B 0.000,C 90.000,E1 273.326} C_DIS
LIN {X 0.042,Y -486.997,Z 655.516,A 0.000,B 0.000,C 90.000,E1 272.808} C_DIS
LIN {X 0.214,Y -487.038,Z 655.513,A 0.000,B 0.000,C 90.000,E1 272.293} C_DIS
LIN {X -0.096,Y -486.798,Z 655.510,A 0.000,B 0.000,C 90.000,E1 271.835} C_DIS
LIN {X 0.094,Y -486.254,Z 655.507,A 0.000,B 0.000,C 90.000,E1 271.318} C_DIS
LIN {X -0.217,Y -485.282,Z 655.505,A 0.000,B 0.000,C 90.000,E1 270.859} C_DIS
LIN {X -0.044,Y -483.813,Z 655.502,A 0.000,B 0.000,C 90.000,E1 270.344} C_DIS
LIN {X 0.122,Y -481.815,Z 655.499,A 0.000,B 0.000,C 90.000,E1 269.828} C_DIS
LIN {X -0.201,Y -479.138,Z 655.496,A 0.000,B 0.000,C 90.000,E1 269.370} C_DIS
LIN {X -0.062,Y -475.698,Z 655.494,A 0.000,B 0.000,C 90.000,E1 268.854} C_DIS
LIN {X -0.240,Y -473.637,Z 655.492,A 0.000,B 0.000,C 90.000,E1 268.625} C_DIS
LIN {X -0.111,Y -468.568,Z 655.489,A 0.000,B 0.000,C 90.000,E1 268.108} C_DIS
LIN {X 0.224,Y -462.650,Z 655.487,A 0.000,B 0.000,C 90.000,E1 267.593} C_DIS
LIN {X 0.137,Y -456.119,Z 655.484,A 0.000,B 0.000,C 90.000,E1 267.192} C_DIS
LIN {X 0.003,Y -452.495,Z 655.483,A 0.000,B 0.000,C 90.000,E1 267.020} C_DIS
LIN {X -0.137,Y -445.128,Z 655.482,A 0.000,B 0.000,C 90.000,E1 266.731} C_DIS
LIN {X 0.207,Y -436.999,Z 655.480,A 0.000,B 0.000,C 90.000,E1 266.445} C_DIS
LIN {X 0.206,Y -428.798,Z 655.479,A 0.000,B 0.000,C 90.000,E1 266.274} C_DIS
LIN {X -0.047,Y -421.366,Z 655.479,A 0.000,B 0.000,C 90.000,E1 266.216} C_DIS
LIN {X 0.089,Y -414.290,Z 655.479,A 0.000,B 0.000,C 90.000,E1 266.159} C_DIS
LIN {X 0.013,Y -180.927,Z 655.479,A 0.000,B 0.000,C 90.000,E1 266.159} C_DIS
LIN {X -0.083,Y -180.902,Z 655.474,A 0.000,B 0.000,C 90.000,E1 265.298} C_DIS
LIN {X 0.046,Y -180.231,Z 655.464,A 0.000,B 0.000,C 90.000,E1 263.571} C_DIS
LIN {X 0.063,Y -178.715,Z 655.441,A 0.000,B 0.000,C 90.000,E1 259.342} C_DIS
LIN {X -0.045,Y -175.763,Z 655.413,A 0.000,B 0.000,C 90.000,E1 254.283} C_DIS
LIN {X 0.005,Y -171.947,Z 655.384,A 0.000,B 0.000,C 90.000,E1 249.135} C_DIS
LIN {X -0.019,Y -171.334,Z 655.379,A 0.000,B 0.000,C 90.000,E1 248.284} C_DIS
LIN {X 0.034,Y -167.588,Z 655.355,A 0.000,B 0.000,C 90.000,E1 243.948} C_DIS
LIN {X -0.028,Y -166.226,Z 655.346,A 0.000,B 0.000,C 90.000,E1 242.231} C_DIS
LIN {X -0.039,Y -162.986,Z 655.326,A 0.000,B 0.000,C 90.000,E1 238.742} C_DIS
LIN {X 0.008,Y -160.904,Z 655.312,A 0.000,B 0.000,C 90.000,E1 236.087} C_DIS
LIN {X -0.014,Y -157.669,Z 655.292,A 0.000,B 0.000,C 90.000,E1 232.557} C_DIS
LIN {X -0.076,Y -155.708,Z 655.277,A 0.000,B 0.000,C 90.000,E1 229.908} C_DIS
LIN {X -0.020,Y -151.970,Z 655.252,A 0.000,B 0.000,C 90.000,E1 225.405} C_DIS
LIN {X -0.005,Y -150.212,Z 655.237,A 0.000,B 0.000,C 90.000,E1 222.690} C_DIS
LIN {X -0.081,Y -146.978,Z 655.212,A 0.000,B 0.000,C 90.000,E1 218.177} C_DIS
LIN {X 0.029,Y -145.565,Z 655.197,A 0.000,B 0.000,C 90.000,E1 215.391} C_DIS
LIN {X 0.028,Y -142.955,Z 655.171,A 0.000,B 0.000,C 90.000,E1 210.797} C_DIS
LIN {X -0.041,Y -141.581,Z 655.151,A 0.000,B 0.000,C 90.000,E1 207.129} C_DIS
LIN {X 0.006,Y -139.417,Z 655.115,A 0.000,B 0.000,C 90.000,E1 200.610} C_DIS
LIN {X 0.058,Y -139.141,Z 655.104,A 0.000,B 0.000,C 90.000,E1 198.725} C_DIS
LIN {X -0.051,Y -138.348,Z 655.057,A 0.000,B 0.000,C 90.000,E1 190.366} C_DIS
LIN {X -0.066,Y -139.491,Z 655.006,A 0.000,B 0.000,C 90.000,E1 181.031} C_DIS
LIN {X 0.014,Y -141.101,Z 654.975,A 0.000,B 0.000,C 90.000,E1 175.412} C_DIS
LIN {X -0.032,Y -142.480,Z 654.959,A 0.000,B 0.000,C 90.000,E1 172.648} C_DIS
LIN {X 0.057,Y -144.728,Z 654.933,A 0.000,B 0.000,C 90.000,E1 167.993} C_DIS
LIN {X 0.008,Y -147.332,Z 654.913,A 0.000,B 0.000,C 90.000,E1 164.338} C_DIS
LIN {X 0.073,Y -150.655,Z 654.888,A 0.000,B 0.000,C 90.000,E1 159.752} C_DIS
LIN {X -0.046,Y -154.133,Z 654.868,A 0.000,B 0.000,C 90.000,E1 156.177} C_DIS
LIN {X 0.017,Y -157.561,Z 654.848,A 0.000,B 0.000,C 90.000,E1 152.564} C_DIS
LIN {X 0.041,Y -161.803,Z 654.828,A 0.000,B 0.000,C 90.000,E1 148.997} C_DIS
LIN {X 0.061,Y -165.995,Z 654.808,A 0.000,B 0.000,C 90.000,E1 145.468} C_DIS
LIN {X 0.054,Y -170.993,Z 654.789,A 0.000,B 0.000,C 90.000,E1 141.984} C_DIS
LIN {X -0.031,Y -175.862,Z 654.770,A 0.000,B 0.000,C 90.000,E1 138.566} C_DIS
LIN {X -0.037,Y -181.468,Z 654.751,A 0.000,B 0.000,C 90.000,E1 135.162} C_DIS
LIN {X 0.100,Y -186.979,Z 654.732,A 0.000,B 0.000,C 90.000,E1 131.757} C_DIS
LIN {X -0.120,Y -191.043,Z 654.720,A 0.000,B 0.000,C 90.000,E1 129.644} C_DIS
LIN {X 0.171,Y -288.630,Z 654.720,A 0.000,B 0.000,C 90.000,E1 129.564} C_DIS
LIN {X 0.015,Y -290.482,Z 654.720,A 0.000,B 0.000,C 90.000,E1 129.564} C_DIS
LIN {X 0.086,Y -295.666,Z 654.718,A 0.000,B 0.000,C 90.000,E1 129.277} C_DIS
LIN {X -0.113,Y -298.857,Z 654.716,A 0.000,B 0.000,C 90.000,E1 128.991} C_DIS
LIN {X 0.059,Y -302.467,Z 654.713,A 0.000,B 0.000,C 90.000,E1 128.382} C_DIS
LIN {X -0.181,Y -303.920,Z 654.711,A 0.000,B 0.000,C 90.000,E1 128.096} C_DIS
LIN {X 0.007,Y -305.063,Z 654.710,A 0.000,B 0.000,C 90.000,E1 127.729} C_DIS
LIN {X 0.117,Y -315.622,Z 654.690,A 0.000,B 0.000,C 90.000,E1 124.119} C_DIS
LIN {X -0.006,Y -325.593,Z 654.674,A 0.000,B 0.000,C 90.000,E1 121.258} C_DIS
LIN {X -0.060,Y -336.884,Z 654.658,A 0.000,B 0.000,C 90.000,E1 118.437} C_DIS
LIN {X -0.107,Y -349.600,Z 654.643,A 0.000,B 0.000,C 90.000,E1 115.668} C_DIS
LIN {X 0.171,Y -362.190,Z 654.629,A 0.000,B 0.000,C 90.000,E1 113.206} C_DIS
LIN {X 0.011,Y -376.084,Z 654.616,A 0.000,B 0.000,C 90.000,E1 110.865} C_DIS
LIN {X 0.062,Y -391.384,Z 654.603,A 0.000,B 0.000,C 90.000,E1 108.544} C_DIS
LIN {X -0.145,Y -408.199,Z 654.591,A 0.000,B 0.000,C 90.000,E1 106.315} C_DIS
LIN {X -0.180,Y -426.654,Z 654.578,A 0.000,B 0.000,C 90.000,E1 104.120} C_DIS
LIN {X -0.114,Y -446.527,Z 654.567,A 0.000,B 0.000,C 90.000,E1 102.007} C_DIS
LIN {X -0.112,Y -467.006,Z 654.556,A 0.000,B 0.000,C 90.000,E1 100.074} C_DIS
LIN {X -0.137,Y -469.589,Z 654.555,A 0.000,B 0.000,C 90.000,E1 99.849} C_DIS
LIN {X -0.081,Y -471.811,Z 654.553,A 0.000,B 0.000,C 90.000,E1 99.613} C_DIS
LIN {X 0.253,Y -473.636,Z 654.552,A 0.000,B 0.000,C 90.000,E1 99.321} C_DIS
LIN {X 0.046,Y -475.009,Z 654.551,A 0.000,B 0.000,C 90.000,E1 99.095} C_DIS
LIN {X 0.240,Y -476.756,Z 654.548,A 0.000,B 0.000,C 90.000,E1 98.568} C_DIS
LIN {X -0.102,Y -477.421,Z 654.545,A 0.000,B 0.000,C 90.000,E1 98.106} C_DIS
LIN {X 0.040,Y -477.118,Z 654.542,A 0.000,B 0.000,C 90.000,E1 97.587} C_DIS
LIN {X 0.187,Y -475.803,Z 654.539,A 0.000,B 0.000,C 90.000,E1 97.068} C_DIS
LIN {X 0.052,Y -474.701,Z 654.538,A 0.000,B 0.000,C 90.000,E1 96.834} C_DIS
LIN {X -0.139,Y -473.226,Z 654.537,A 0.000,B 0.000,C 90.000,E1 96.606} C_DIS
LIN {X -0.151,Y -456.154,Z 654.523,A 0.000,B 0.000,C 90.000,E1 94.069} C_DIS
LIN {X 0.012,Y -445.459,Z 654.512,A 0.000,B 0.000,C 90.000,E1 92.236} C_DIS
LIN {X -0.028,Y -435.404,Z 654.502,A 0.000,B 0.000,C 90.000,E1 90.401} C_DIS
LIN {X -0.128,Y -427.999,Z 654.495,A 0.000,B 0.000,C 90.000,E1 89.083} C_DIS
LIN {X -0.205,Y -418.743,Z 654.486,A 0.000,B 0.000,C 90.000,E1 87.478} C_DIS
LIN {X -0.006,Y -409.357,Z 654.477,A 0.000,B 0.000,C 90.000,E1 85.812} C_DIS
LIN {X -0.185,Y -395.550,Z 654.463,A 0.000,B 0.000,C 90.000,E1 83.337} C_DIS
LIN {X 0.133,Y -382.204,Z 654.449,A 0.000,B 0.000,C 90.000,E1 80.735} C_DIS
LIN {X -0.164,Y -369.365,Z 654.434,A 0.000,B 0.000,C 90.000,E1 78.173} C_DIS
LIN {X 0.142,Y -356.988,Z 654.419,A 0.000,B 0.000,C 90.000,E1 75.463} C_DIS
LIN {X -0.044,Y -345.288,Z 654.404,A 0.000,B 0.000,C 90.000,E1 72.779} C_DIS
LIN {X -0.064,Y -330.638,Z 654.384,A 0.000,B 0.000,C 90.000,E1 69.082} C_DIS
LIN {X -0.005,Y -317.319,Z 654.363,A 0.000,B 0.000,C 90.000,E1 65.281} C_DIS
LIN {X 0.129,Y -305.517,Z 654.341,A 0.000,B 0.000,C 90.000,E1 61.385} C_DIS
LIN {X 0.024,Y -294.933,Z 654.319,A 0.000,B 0.000,C 90.000,E1 57.454} C_DIS
LIN {X 0.074,Y -288.302,Z 654.304,A 0.000,B 0.000,C 90.000,E1 54.769} C_DIS
LIN {X 0.052,Y -281.896,Z 654.289,A 0.000,B 0.000,C 90.000,E1 52.065} C_DIS
LIN {X -0.049,Y -276.873,Z 654.278,A 0.000,B 0.000,C 90.000,E1 50.033} C_DIS
LIN {X -0.031,Y -271.405,Z 654.266,A 0.000,B 0.000,C 90.000,E1 47.957} C_DIS
LIN {X -0.155,Y -265.529,Z 654.255,A 0.000,B 0.000,C 90.000,E1 45.891} C_DIS
LIN {X -0.012,Y -259.240,Z 654.243,A 0.000,B 0.000,C 90.000,E1 43.743} C_DIS
LIN {X 0.010,Y -252.679,Z 654.231,A 0.000,B 0.000,C 90.000,E1 41.595} C_DIS
LIN {X -0.027,Y -241.914,Z 654.211,A 0.000,B 0.000,C 90.000,E1 37.971} C_DIS
LIN {X -0.097,Y -233.951,Z 654.194,A 0.000,B 0.000,C 90.000,E1 35.025} C_DIS
LIN {X 0.081,Y -224.947,Z 654.174,A 0.000,B 0.000,C 90.000,E1 31.209} C_DIS
LIN {X 0.038,Y -218.600,Z 654.156,A 0.000,B 0.000,C 90.000,E1 28.153} C_DIS
LIN {X -0.086,Y -213.094,Z 654.139,A 0.000,B 0.000,C 90.000,E1 25.079} C_DIS
LIN {X 0.080,Y -207.266,Z 654.117,A 0.000,B 0.000,C 90.000,E1 21.099} C_DIS
LIN {X -0.036,Y -202.599,Z 654.095,A 0.000,B 0.000,C 90.000,E1 17.149} C_DIS
LIN {X -0.005,Y -199.037,Z 654.073,A 0.000,B 0.000,C 90.000,E1 13.119} C_DIS
LIN {X 0.104,Y -195.681,Z 654.041,A 0.000,B 0.000,C 90.000,E1 7.409} C_DIS
LIN {X -0.020,Y -196.508,Z 653.957,A 0.000,B 0.000,C 90.000,E1 352.186} C_DIS
LIN {X 0.029,Y -199.778,Z 653.930,A 0.000,B 0.000,C 90.000,E1 347.297} C_DIS
LIN {X 0.016,Y -203.573,Z 653.907,A 0.000,B 0.000,C 90.000,E1 343.268} C_DIS
LIN {X 0.043,Y -208.358,Z 653.885,A 0.000,B 0.000,C 90.000,E1 339.263} C_DIS
LIN {X 0.054,Y -213.952,Z 653.863,A 0.000,B 0.000,C 90.000,E1 335.305} C_DIS
LIN {X 0.105,Y -220.275,Z 653.841,A 0.000,B 0.000,C 90.000,E1 331.385} C_DIS
LIN {X -0.015,Y -225.833,Z 653.824,A 0.000,B 0.000,C 90.000,E1 328.329} C_DIS
LIN {X -0.051,Y -233.194,Z 653.803,A 0.000,B 0.000,C 90.000,E1 324.529} C_DIS
LIN {X -0.157,Y -241.202,Z 653.782,A 0.000,B 0.000,C 90.000,E1 320.803} C_DIS
LIN {X 0.045,Y -250.037,Z 653.762,A 0.000,B 0.000,C 90.000,E1 317.067} C_DIS
LIN {X -0.021,Y -259.862,Z 653.741,A 0.000,B 0.000,C 90.000,E1 313.461} C_DIS
LIN {X -0.035,Y -268.619,Z 653.726,A 0.000,B 0.000,C 90.000,E1 310.620} C_DIS
LIN {X -0.132,Y -281.027,Z 653.706,A 0.000,B 0.000,C 90.000,E1 307.156} C_DIS
LIN {X 0.118,Y -294.752,Z 653.687,A 0.000,B 0.000,C 90.000,E1 303.706} C_DIS
LIN {X -0.022,Y -308.568,Z 653.671,A 0.000,B 0.000,C 90.000,E1 300.747} C_DIS
LIN {X 0.002,Y -325.287,Z 653.653,A 0.000,B 0.000,C 90.000,E1 297.513} C_DIS
LIN {X -0.180,Y -339.233,Z 653.639,A 0.000,B 0.000,C 90.000,E1 295.027} C_DIS
LIN {X 0.191,Y -355.746,Z 653.624,A 0.000,B 0.000,C 90.000,E1 292.206} C_DIS
LIN {X 0.143,Y -369.308,Z 653.612,A 0.000,B 0.000,C 90.000,E1 290.120} C_DIS
LIN {X -0.102,Y -384.342,Z 653.601,A 0.000,B 0.000,C 90.000,E1 288.109} C_DIS
LIN {X 0.176,Y -402.918,Z 653.588,A 0.000,B 0.000,C 90.000,E1 285.788} C_DIS
LIN {X -0.035,Y -414.510,Z 653.580,A 0.000,B 0.000,C 90.000,E1 284.426} C_DIS
LIN {X -0.088,Y -425.622,Z 653.573,A 0.000,B 0.000,C 90.000,E1 283.063} C_DIS
LIN {X -0.068,Y -436.194,Z 653.565,A 0.000,B 0.000,C 90.000,E1 281.715} C_DIS
LIN {X -0.118,Y -444.326,Z 653.559,A 0.000,B 0.000,C 90.000,E1 280.658} C_DIS
LIN {X 0.087,Y -454.209,Z 653.552,A 0.000,B 0.000,C 90.000,E1 279.321} C_DIS
LIN {X 0.090,Y -464.887,Z 653.545,A 0.000,B 0.000,C 90.000,E1 278.049} C_DIS
LIN {X -0.015,Y -470.623,Z 653.541,A 0.000,B 0.000,C 90.000,E1 277.296} C_DIS
LIN {X -0.070,Y -475.426,Z 653.536,A 0.000,B 0.000,C 90.000,E1 276.543} C_DIS
LIN {X -0.142,Y -479.430,Z 653.532,A 0.000,B 0.000,C 90.000,E1 275.796} C_DIS
LIN {X 0.009,Y -481.613,Z 653.529,A 0.000,B 0.000,C 90.000,E1 275.277} C_DIS
LIN {X 0.174,Y -483.483,Z 653.527,A 0.000,B 0.000,C 90.000,E1 274.759} C_DIS
LIN {X -0.177,Y -484.908,Z 653.524,A 0.000,B 0.000,C 90.000,E1 274.302} C_DIS
LIN {X 0.003,Y -485.950,Z 653.521,A 0.000,B 0.000,C 90.000,E1 273.784} C_DIS
LIN {X 0.161,Y -486.607,Z 653.518,A 0.000,B 0.000,C 90.000,E1 273.269} C_DIS
LIN {X -0.133,Y -486.922,Z 653.516,A 0.000,B 0.000,C 90.000,E1 272.808} C_DIS
LIN {X 0.038,Y -486.998,Z 653.513,A 0.000,B 0.000,C 90.000,E1 272.293} C_DIS
LIN {X 0.229,Y -486.745,Z 653.510,A 0.000,B 0.000,C 90.000,E1 271.776} C_DIS
LIN {X -0.082,Y -486.167,Z 653.507,A 0.000,B 0.000,C 90.000,E1 271.318} C_DIS
LIN {X 0.092,Y -485.187,Z 653.505,A 0.000,B 0.000,C 90.000,E1 270.802} C_DIS
LIN {X -0.220,Y -483.717,Z 653.502,A 0.000,B 0.000,C 90.000,E1 270.344} C_DIS
LIN {X -0.053,Y -481.684,Z 653.499,A 0.000,B 0.000,C 90.000,E1 269.828} C_DIS
LIN {X 0.103,Y -479.025,Z 653.496,A 0.000,B 0.000,C 90.000,E1 269.312} C_DIS
LIN {X -0.237,Y -475.551,Z 653.493,A 0.000,B 0.000,C 90.000,E1 268.854} C_DIS
LIN {X -0.119,Y -471.000,Z 653.491,A 0.000,B 0.000,C 90.000,E1 268.339} C_DIS
LIN {X 0.178,Y -468.373,Z 653.489,A 0.000,B 0.000,C 90.000,E1 268.051} C_DIS
LIN {X -0.009,Y -465.364,Z 653.488,A 0.000,B 0.000,C 90.000,E1 267.822} C_DIS
LIN {X 0.115,Y -459.045,Z 653.485,A 0.000,B 0.000,C 90.000,E1 267.364} C_DIS
LIN {X -0.012,Y -455.873,Z 653.484,A 0.000,B 0.000,C 90.000,E1 267.192} C_DIS
LIN {X 0.051,Y -448.813,Z 653.482,A 0.000,B 0.000,C 90.000,E1 266.846} C_DIS
